Yaskawa INFORM job: DEMO_ROOF_SIDE_0625_3PAINT_3.JBI

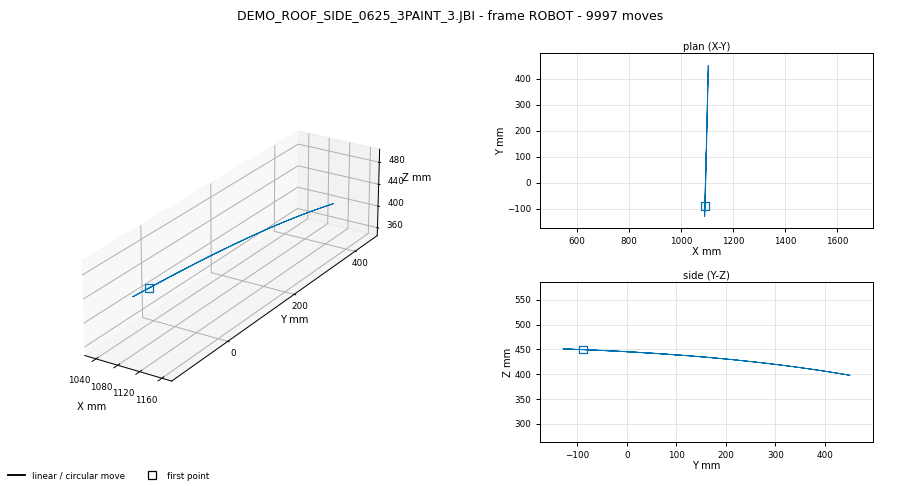
[picture p0: tool path of DEMO_ROOF_SIDE_0625_3PAINT_3.JBI in frame ROBOT, 9997 of 9997 moves have a stored position in this frame; points joined in program order, loops and branches not executed]
/JOB
//NAME DEMO_ROOF_SIDE_0625_3PAINT3
//POS
///NPOS 9997,0,0,0,0,0
///TOOL 0
///USER 0
///POSTYPE ROBOT
///RECTAN
///RCONF 1,0,0,0,0,0,0,0,0,0,0,0,0,0,0,0,0,0,0,0,0,0,0,0
C00000=1093.396,-88.065,450.012,175.022,15.482,152.318
C00001=1093.401,-87.815,450.002,175.023,15.482,152.318
C00002=1093.408,-87.566,449.991,175.025,15.483,152.317
C00003=1093.413,-87.316,449.981,175.027,15.484,152.317
C00004=1093.419,-87.066,449.970,175.029,15.485,152.317
C00005=1093.425,-86.817,449.960,175.030,15.485,152.317
C00006=1093.432,-86.567,449.949,175.032,15.486,152.317
C00007=1093.438,-86.317,449.939,175.033,15.487,152.316
C00008=1093.444,-86.068,449.928,175.035,15.487,152.316
C00009=1093.449,-85.818,449.918,175.037,15.488,152.316
C00010=1093.456,-85.568,449.908,175.038,15.488,152.316
C00011=1093.462,-85.318,449.897,175.040,15.489,152.316
C00012=1093.468,-85.069,449.886,175.042,15.490,152.315
C00013=1093.474,-84.819,449.876,175.044,15.491,152.315
C00014=1093.480,-84.569,449.865,175.045,15.491,152.315
C00015=1093.486,-84.320,449.855,175.046,15.492,152.315
C00016=1093.492,-84.070,449.844,175.048,15.493,152.315
C00017=1093.499,-83.820,449.834,175.050,15.493,152.314
C00018=1093.504,-83.571,449.823,175.052,15.494,152.314
C00019=1093.510,-83.321,449.813,175.053,15.495,152.314
C00020=1093.517,-83.071,449.803,175.055,15.495,152.314
C00021=1093.523,-82.821,449.792,175.057,15.496,152.313
C00022=1093.528,-82.572,449.781,175.059,15.497,152.313
C00023=1093.535,-82.322,449.771,175.060,15.498,152.313
C00024=1093.541,-82.072,449.759,175.061,15.498,152.313
C00025=1093.547,-81.822,449.750,175.063,15.499,152.313
C00026=1093.553,-81.573,449.739,175.065,15.499,152.312
C00027=1093.559,-81.323,449.728,175.067,15.500,152.312
C00028=1093.566,-81.050,449.716,175.069,15.501,152.312
C00029=1093.573,-80.778,449.704,175.070,15.502,152.312
C00030=1093.579,-80.506,449.693,175.072,15.502,152.311
C00031=1093.585,-80.233,449.682,175.074,15.504,152.311
C00032=1093.591,-79.984,449.671,175.075,15.504,152.311
C00033=1093.598,-79.734,449.660,175.077,15.504,152.311
C00034=1093.604,-79.484,449.650,175.079,15.505,152.311
C00035=1093.610,-79.235,449.639,175.080,15.506,152.310
C00036=1093.615,-78.985,449.628,175.082,15.507,152.310
C00037=1093.621,-78.734,449.617,175.084,15.508,152.310
C00038=1093.628,-78.485,449.607,175.085,15.508,152.310
C00039=1093.634,-78.236,449.596,175.087,15.509,152.310
C00040=1093.639,-77.986,449.585,175.088,15.510,152.309
C00041=1093.646,-77.736,449.574,175.090,15.511,152.309
C00042=1093.652,-77.487,449.563,175.092,15.511,152.309
C00043=1093.657,-77.236,449.553,175.094,15.513,152.309
C00044=1093.663,-76.987,449.543,175.095,15.513,152.309
C00045=1093.670,-76.737,449.531,175.097,15.513,152.308
C00046=1093.676,-76.488,449.521,175.098,15.515,152.308
C00047=1093.681,-76.238,449.510,175.100,15.515,152.308
C00048=1093.687,-75.989,449.499,175.102,15.516,152.308
C00049=1093.693,-75.738,449.488,175.104,15.517,152.308
C00050=1093.700,-75.489,449.477,175.105,15.517,152.307
C00051=1093.706,-75.240,449.466,175.106,15.518,152.307
C00052=1093.712,-74.990,449.455,175.108,15.519,152.307
C00053=1093.718,-74.740,449.444,175.110,15.520,152.307
C00054=1093.723,-74.491,449.433,175.112,15.521,152.307
C00055=1093.729,-74.241,449.422,175.114,15.522,152.306
C00056=1093.735,-73.991,449.411,175.116,15.522,152.306
C00057=1093.741,-73.741,449.401,175.116,15.523,152.306
C00058=1093.747,-73.491,449.390,175.118,15.523,152.306
C00059=1093.752,-73.242,449.379,175.120,15.525,152.306
C00060=1093.759,-72.992,449.368,175.122,15.525,152.305
C00061=1093.764,-72.742,449.357,175.123,15.526,152.305
C00062=1093.770,-72.493,449.346,175.125,15.527,152.305
C00063=1093.776,-72.243,449.335,175.127,15.528,152.305
C00064=1093.782,-71.993,449.324,175.128,15.528,152.305
C00065=1093.788,-71.743,449.313,175.130,15.530,152.305
C00066=1093.794,-71.494,449.302,175.132,15.530,152.304
C00067=1093.799,-71.245,449.292,175.133,15.531,152.304
C00068=1093.806,-70.994,449.280,175.135,15.532,152.304
C00069=1093.812,-70.745,449.269,175.137,15.533,152.304
C00070=1093.818,-70.496,449.258,175.138,15.534,152.304
C00071=1093.824,-70.246,449.247,175.140,15.535,152.303
C00072=1093.830,-69.996,449.236,175.141,15.535,152.303
C00073=1093.835,-69.746,449.224,175.143,15.536,152.303
C00074=1093.840,-69.497,449.213,175.145,15.537,152.303
C00075=1093.847,-69.247,449.202,175.147,15.538,152.303
C00076=1093.853,-68.997,449.191,175.148,15.539,152.303
C00077=1093.858,-68.748,449.180,175.150,15.540,152.302
C00078=1093.865,-68.498,449.169,175.152,15.541,152.302
C00079=1093.870,-68.248,449.158,175.154,15.541,152.302
C00080=1093.876,-67.999,449.147,175.155,15.543,152.302
C00081=1093.882,-67.748,449.136,175.156,15.543,152.302
C00082=1093.888,-67.500,449.125,175.158,15.543,152.301
C00083=1093.894,-67.250,449.114,175.160,15.545,152.301
C00084=1093.900,-67.000,449.102,175.162,15.545,152.301
C00085=1093.906,-66.750,449.091,175.163,15.546,152.301
C00086=1093.911,-66.501,449.080,175.165,15.547,152.301
C00087=1093.918,-66.250,449.069,175.167,15.548,152.300
C00088=1093.923,-66.001,449.058,175.169,15.549,152.300
C00089=1093.929,-65.752,449.046,175.170,15.550,152.300
C00090=1093.936,-65.502,449.035,175.171,15.550,152.300
C00091=1093.941,-65.252,449.024,175.173,15.551,152.300
C00092=1093.948,-64.982,449.012,175.175,15.552,152.300
C00093=1093.954,-64.711,449.000,175.177,15.554,152.299
C00094=1093.960,-64.441,448.988,175.179,15.555,152.299
C00095=1093.967,-64.171,448.975,175.181,15.555,152.299
C00096=1093.972,-63.921,448.964,175.182,15.556,152.299
C00097=1093.979,-63.672,448.952,175.184,15.556,152.299
C00098=1093.985,-63.422,448.942,175.185,15.558,152.298
C00099=1093.991,-63.172,448.930,175.187,15.558,152.298
C00100=1093.997,-62.922,448.919,175.189,15.559,152.298
C00101=1094.002,-62.673,448.907,175.191,15.560,152.298
C00102=1094.009,-62.423,448.896,175.192,15.561,152.298
C00103=1094.014,-62.174,448.885,175.194,15.562,152.297
C00104=1094.021,-61.923,448.874,175.196,15.563,152.297
C00105=1094.027,-61.674,448.862,175.198,15.564,152.297
C00106=1094.033,-61.424,448.851,175.199,15.565,152.297
C00107=1094.038,-61.174,448.840,175.201,15.566,152.297
C00108=1094.044,-60.926,448.828,175.203,15.567,152.297
C00109=1094.050,-60.675,448.817,175.204,15.567,152.296
C00110=1094.056,-60.426,448.806,175.205,15.568,152.296
C00111=1094.063,-60.176,448.795,175.207,15.569,152.296
C00112=1094.068,-59.927,448.782,175.209,15.570,152.296
C00113=1094.074,-59.676,448.771,175.211,15.571,152.296
C00114=1094.080,-59.427,448.760,175.213,15.571,152.295
C00115=1094.087,-59.177,448.748,175.214,15.573,152.295
C00116=1094.092,-58.928,448.738,175.216,15.573,152.295
C00117=1094.098,-58.677,448.726,175.218,15.574,152.295
C00118=1094.104,-58.428,448.714,175.220,15.575,152.295
C00119=1094.110,-58.178,448.703,175.221,15.576,152.295
C00120=1094.116,-57.929,448.691,175.223,15.577,152.294
C00121=1094.123,-57.679,448.680,175.225,15.578,152.294
C00122=1094.128,-57.429,448.669,175.226,15.579,152.294
C00123=1094.134,-57.181,448.657,175.228,15.580,152.294
C00124=1094.140,-56.930,448.646,175.230,15.581,152.294
C00125=1094.147,-56.681,448.634,175.231,15.581,152.294
C00126=1094.152,-56.431,448.622,175.233,15.582,152.293
C00127=1094.158,-56.181,448.611,175.234,15.583,152.293
C00128=1094.164,-55.932,448.599,175.236,15.584,152.293
C00129=1094.170,-55.682,448.588,175.238,15.585,152.293
C00130=1094.176,-55.433,448.576,175.240,15.586,152.293
C00131=1094.182,-55.182,448.565,175.241,15.587,152.292
C00132=1094.188,-54.933,448.553,175.243,15.588,152.292
C00133=1094.194,-54.683,448.542,175.245,15.589,152.292
C00134=1094.200,-54.434,448.530,175.247,15.589,152.292
C00135=1094.206,-54.184,448.519,175.248,15.590,152.292
C00136=1094.212,-53.935,448.507,175.250,15.591,152.291
C00137=1094.218,-53.685,448.496,175.252,15.592,152.291
C00138=1094.224,-53.436,448.483,175.254,15.593,152.291
C00139=1094.230,-53.185,448.472,175.255,15.594,152.291
C00140=1094.237,-52.936,448.460,175.257,15.595,152.291
C00141=1094.243,-52.686,448.449,175.259,15.596,152.290
C00142=1094.248,-52.437,448.437,175.261,15.597,152.290
C00143=1094.254,-52.187,448.426,175.262,15.597,152.290
C00144=1094.261,-51.937,448.414,175.264,15.599,152.290
C00145=1094.266,-51.687,448.402,175.266,15.599,152.290
C00146=1094.272,-51.438,448.391,175.267,15.600,152.290
C00147=1094.279,-51.188,448.379,175.269,15.601,152.289
C00148=1094.284,-50.939,448.367,175.270,15.602,152.289
C00149=1094.291,-50.689,448.355,175.272,15.602,152.289
C00150=1094.297,-50.439,448.344,175.274,15.604,152.289
C00151=1094.302,-50.190,448.332,175.276,15.604,152.289
C00152=1094.309,-49.940,448.321,175.277,15.605,152.289
C00153=1094.314,-49.690,448.308,175.279,15.606,152.288
C00154=1094.321,-49.441,448.296,175.281,15.607,152.288
C00155=1094.326,-49.191,448.285,175.282,15.609,152.288
C00156=1094.332,-48.922,448.272,175.285,15.610,152.288
C00157=1094.338,-48.653,448.259,175.286,15.611,152.288
C00158=1094.345,-48.384,448.247,175.288,15.612,152.287
C00159=1094.351,-48.115,448.234,175.290,15.613,152.287
C00160=1094.357,-47.866,448.222,175.292,15.613,152.287
C00161=1094.363,-47.615,448.211,175.293,15.615,152.287
C00162=1094.368,-47.366,448.198,175.295,15.615,152.287
C00163=1094.375,-47.117,448.187,175.297,15.617,152.287
C00164=1094.381,-46.866,448.175,175.299,15.618,152.286
C00165=1094.386,-46.617,448.162,175.300,15.618,152.286
C00166=1094.393,-46.367,448.151,175.302,15.620,152.286
C00167=1094.398,-46.118,448.138,175.304,15.620,152.286
C00168=1094.404,-45.868,448.127,175.305,15.621,152.286
C00169=1094.410,-45.618,448.115,175.307,15.622,152.286
C00170=1094.416,-45.369,448.103,175.309,15.623,152.285
C00171=1094.422,-45.119,448.091,175.311,15.624,152.285
C00172=1094.427,-44.870,448.079,175.312,15.625,152.285
C00173=1094.434,-44.620,448.067,175.314,15.626,152.285
C00174=1094.440,-44.370,448.054,175.316,15.627,152.285
C00175=1094.445,-44.121,448.044,175.318,15.628,152.285
C00176=1094.451,-43.871,448.031,175.319,15.629,152.284
C00177=1094.457,-43.622,448.019,175.321,15.630,152.284
C00178=1094.463,-43.372,448.007,175.323,15.631,152.284
C00179=1094.469,-43.122,447.995,175.324,15.632,152.284
C00180=1094.475,-42.873,447.983,175.326,15.633,152.284
C00181=1094.481,-42.623,447.971,175.328,15.634,152.284
C00182=1094.487,-42.373,447.959,175.330,15.635,152.283
C00183=1094.492,-42.123,447.947,175.331,15.636,152.283
C00184=1094.498,-41.874,447.935,175.333,15.637,152.283
C00185=1094.504,-41.625,447.923,175.335,15.638,152.283
C00186=1094.510,-41.375,447.911,175.337,15.639,152.283
C00187=1094.516,-41.125,447.898,175.338,15.640,152.283
C00188=1094.522,-40.876,447.887,175.340,15.641,152.282
C00189=1094.528,-40.626,447.875,175.342,15.642,152.282
C00190=1094.535,-40.376,447.863,175.343,15.642,152.282
C00191=1094.540,-40.126,447.850,175.345,15.644,152.282
C00192=1094.546,-39.877,447.838,175.347,15.644,152.282
C00193=1094.552,-39.627,447.826,175.349,15.645,152.281
C00194=1094.558,-39.377,447.814,175.351,15.647,152.281
C00195=1094.564,-39.128,447.801,175.353,15.648,152.281
C00196=1094.570,-38.878,447.790,175.354,15.649,152.281
C00197=1094.576,-38.628,447.778,175.356,15.650,152.281
C00198=1094.581,-38.379,447.765,175.358,15.651,152.281
C00199=1094.587,-38.129,447.753,175.360,15.652,152.280
C00200=1094.594,-37.880,447.741,175.361,15.653,152.280
C00201=1094.599,-37.630,447.729,175.363,15.654,152.280
C00202=1094.605,-37.381,447.716,175.365,15.655,152.280
C00203=1094.611,-37.131,447.704,175.366,15.656,152.280
C00204=1094.616,-36.881,447.691,175.368,15.657,152.280
C00205=1094.622,-36.632,447.679,175.370,15.658,152.279
C00206=1094.629,-36.382,447.667,175.372,15.659,152.279
C00207=1094.634,-36.133,447.655,175.373,15.659,152.279
C00208=1094.640,-35.883,447.642,175.375,15.661,152.279
C00209=1094.646,-35.633,447.630,175.377,15.662,152.279
C00210=1094.651,-35.384,447.617,175.378,15.663,152.279
C00211=1094.658,-35.134,447.605,175.380,15.664,152.279
C00212=1094.664,-34.884,447.593,175.382,15.664,152.278
C00213=1094.669,-34.635,447.581,175.384,15.666,152.278
C00214=1094.675,-34.385,447.568,175.386,15.667,152.278
C00215=1094.681,-34.135,447.556,175.388,15.668,152.278
C00216=1094.687,-33.886,447.543,175.389,15.669,152.278
C00217=1094.692,-33.636,447.531,175.391,15.670,152.277
C00218=1094.699,-33.387,447.519,175.393,15.671,152.277
C00219=1094.705,-33.137,447.506,175.394,15.672,152.277
C00220=1094.711,-32.868,447.493,175.396,15.673,152.277
C00221=1094.718,-32.600,447.479,175.398,15.674,152.277
C00222=1094.722,-32.331,447.467,175.401,15.675,152.277
C00223=1094.729,-32.062,447.453,175.402,15.677,152.276
C00224=1094.735,-31.812,447.441,175.404,15.677,152.276
C00225=1094.742,-31.563,447.428,175.406,15.678,152.276
C00226=1094.748,-31.313,447.415,175.407,15.680,152.276
C00227=1094.753,-31.064,447.403,175.409,15.680,152.276
C00228=1094.759,-30.814,447.391,175.411,15.681,152.276
C00229=1094.765,-30.564,447.378,175.413,15.682,152.275
C00230=1094.771,-30.315,447.366,175.414,15.683,152.275
C00231=1094.777,-30.065,447.353,175.416,15.684,152.275
C00232=1094.782,-29.816,447.341,175.419,15.686,152.275
C00233=1094.788,-29.566,447.328,175.420,15.687,152.275
C00234=1094.794,-29.316,447.315,175.422,15.688,152.275
C00235=1094.801,-29.067,447.303,175.424,15.689,152.274
C00236=1094.807,-28.817,447.290,175.426,15.689,152.274
C00237=1094.812,-28.568,447.278,175.427,15.691,152.274
C00238=1094.818,-28.318,447.266,175.429,15.692,152.274
C00239=1094.824,-28.069,447.252,175.431,15.693,152.274
C00240=1094.830,-27.819,447.240,175.432,15.694,152.274
C00241=1094.836,-27.569,447.227,175.434,15.694,152.273
C00242=1094.841,-27.320,447.215,175.436,15.696,152.273
C00243=1094.847,-27.070,447.203,175.438,15.696,152.273
C00244=1094.853,-26.820,447.189,175.440,15.698,152.273
C00245=1094.859,-26.571,447.177,175.442,15.699,152.273
C00246=1094.865,-26.321,447.164,175.443,15.700,152.272
C00247=1094.870,-26.072,447.152,175.445,15.701,152.272
C00248=1094.877,-25.822,447.139,175.447,15.702,152.272
C00249=1094.882,-25.572,447.126,175.448,15.703,152.272
C00250=1094.888,-25.323,447.114,175.450,15.704,152.272
C00251=1094.894,-25.072,447.101,175.452,15.705,152.272
C00252=1094.899,-24.824,447.088,175.454,15.706,152.272
C00253=1094.905,-24.574,447.075,175.456,15.708,152.271
C00254=1094.911,-24.324,447.063,175.458,15.708,152.271
C00255=1094.917,-24.074,447.050,175.459,15.710,152.271
C00256=1094.923,-23.825,447.037,175.461,15.710,152.271
C00257=1094.929,-23.575,447.024,175.463,15.711,152.271
C00258=1094.934,-23.326,447.012,175.464,15.713,152.271
C00259=1094.940,-23.077,446.999,175.466,15.713,152.270
C00260=1094.946,-22.826,446.986,175.468,15.714,152.270
C00261=1094.952,-22.576,446.973,175.470,15.715,152.270
C00262=1094.958,-22.327,446.960,175.472,15.717,152.270
C00263=1094.964,-22.077,446.947,175.474,15.718,152.270
C00264=1094.969,-21.828,446.935,175.476,15.719,152.270
C00265=1094.975,-21.579,446.922,175.477,15.720,152.269
C00266=1094.981,-21.329,446.909,175.479,15.721,152.269
C00267=1094.987,-21.079,446.895,175.481,15.722,152.269
C00268=1094.993,-20.829,446.883,175.482,15.723,152.269
C00269=1094.998,-20.580,446.870,175.484,15.724,152.269
C00270=1095.005,-20.330,446.857,175.487,15.725,152.269
C00271=1095.011,-20.080,446.844,175.489,15.726,152.268
C00272=1095.016,-19.832,446.831,175.490,15.727,152.268
C00273=1095.021,-19.582,446.818,175.492,15.729,152.268
C00274=1095.027,-19.332,446.806,175.494,15.729,152.268
C00275=1095.033,-19.083,446.792,175.495,15.730,152.268
C00276=1095.039,-18.833,446.780,175.497,15.731,152.267
C00277=1095.046,-18.583,446.767,175.499,15.732,152.267
C00278=1095.051,-18.334,446.754,175.501,15.734,152.267
C00279=1095.057,-18.084,446.740,175.503,15.735,152.267
C00280=1095.063,-17.834,446.728,175.505,15.736,152.267
C00281=1095.069,-17.585,446.714,175.506,15.737,152.267
C00282=1095.075,-17.335,446.702,175.508,15.738,152.267
C00283=1095.081,-17.086,446.689,175.510,15.738,152.266
C00284=1095.087,-16.817,446.675,175.512,15.740,152.266
C00285=1095.093,-16.547,446.660,175.514,15.741,152.266
C00286=1095.100,-16.277,446.646,175.516,15.742,152.266
C00287=1095.106,-16.007,446.632,175.518,15.743,152.266
C00288=1095.112,-15.758,446.619,175.520,15.745,152.265
C00289=1095.118,-15.509,446.606,175.522,15.745,152.265
C00290=1095.124,-15.259,446.593,175.524,15.746,152.265
C00291=1095.129,-15.010,446.580,175.525,15.747,152.265
C00292=1095.135,-14.760,446.567,175.527,15.748,152.265
C00293=1095.141,-14.511,446.554,175.529,15.749,152.265
C00294=1095.146,-14.260,446.541,175.531,15.751,152.264
C00295=1095.152,-14.011,446.527,175.533,15.752,152.264
C00296=1095.159,-13.762,446.514,175.535,15.753,152.264
C00297=1095.164,-13.512,446.501,175.536,15.754,152.264
C00298=1095.170,-13.262,446.488,175.538,15.755,152.264
C00299=1095.175,-13.012,446.475,175.540,15.756,152.263
C00300=1095.181,-12.763,446.461,175.541,15.757,152.263
C00301=1095.188,-12.514,446.448,175.544,15.758,152.263
C00302=1095.193,-12.264,446.435,175.546,15.759,152.263
C00303=1095.199,-12.014,446.422,175.547,15.760,152.263
C00304=1095.204,-11.765,446.408,175.549,15.761,152.263
C00305=1095.210,-11.515,446.395,175.551,15.762,152.263
C00306=1095.217,-11.266,446.382,175.553,15.763,152.262
C00307=1095.222,-11.016,446.368,175.555,15.765,152.262
C00308=1095.228,-10.766,446.356,175.557,15.765,152.262
C00309=1095.233,-10.516,446.342,175.559,15.767,152.262
C00310=1095.240,-10.267,446.328,175.560,15.768,152.262
C00311=1095.245,-10.017,446.315,175.562,15.768,152.261
C00312=1095.251,-9.768,446.302,175.564,15.770,152.261
C00313=1095.257,-9.519,446.289,175.566,15.771,152.261
C00314=1095.262,-9.268,446.276,175.568,15.772,152.261
C00315=1095.269,-9.019,446.262,175.570,15.773,152.261
C00316=1095.274,-8.769,446.248,175.571,15.774,152.261
C00317=1095.280,-8.520,446.235,175.573,15.775,152.260
C00318=1095.285,-8.270,446.222,175.576,15.776,152.260
C00319=1095.292,-8.021,446.209,175.577,15.778,152.260
C00320=1095.297,-7.771,446.195,175.579,15.778,152.260
C00321=1095.303,-7.522,446.182,175.581,15.779,152.260
C00322=1095.309,-7.272,446.168,175.583,15.780,152.259
C00323=1095.315,-7.022,446.155,175.584,15.781,152.259
C00324=1095.321,-6.773,446.142,175.587,15.783,152.259
C00325=1095.326,-6.524,446.128,175.588,15.784,152.259
C00326=1095.333,-6.274,446.115,175.590,15.785,152.259
C00327=1095.338,-6.025,446.101,175.592,15.786,152.259
C00328=1095.344,-5.775,446.088,175.594,15.786,152.258
C00329=1095.350,-5.525,446.075,175.595,15.788,152.258
C00330=1095.356,-5.276,446.061,175.598,15.789,152.258
C00331=1095.362,-5.026,446.047,175.600,15.790,152.258
C00332=1095.368,-4.777,446.034,175.602,15.791,152.258
C00333=1095.373,-4.527,446.020,175.603,15.792,152.258
C00334=1095.380,-4.278,446.007,175.605,15.793,152.257
C00335=1095.385,-4.028,445.993,175.607,15.794,152.257
C00336=1095.391,-3.778,445.980,175.609,15.795,152.257
C00337=1095.397,-3.529,445.966,175.611,15.796,152.257
C00338=1095.402,-3.279,445.952,175.613,15.797,152.257
C00339=1095.408,-3.030,445.939,175.614,15.798,152.256
C00340=1095.414,-2.780,445.925,175.617,15.799,152.256
C00341=1095.419,-2.531,445.911,175.619,15.801,152.256
C00342=1095.425,-2.281,445.898,175.620,15.802,152.256
C00343=1095.431,-2.031,445.884,175.622,15.802,152.256
C00344=1095.437,-1.782,445.870,175.624,15.804,152.256
C00345=1095.442,-1.532,445.856,175.626,15.805,152.255
C00346=1095.449,-1.283,445.843,175.628,15.806,152.255
C00347=1095.454,-1.033,445.829,175.630,15.807,152.255
C00348=1095.460,-0.762,445.815,175.631,15.808,152.255
C00349=1095.466,-0.491,445.799,175.634,15.809,152.255
C00350=1095.472,-0.220,445.785,175.636,15.810,152.254
C00351=1095.478,0.052,445.770,175.638,15.812,152.254
C00352=1095.485,0.302,445.756,175.640,15.813,152.254
C00353=1095.490,0.551,445.743,175.642,15.814,152.254
C00354=1095.496,0.801,445.729,175.644,15.815,152.254
C00355=1095.502,1.050,445.714,175.646,15.816,152.254
C00356=1095.508,1.299,445.701,175.648,15.817,152.253
C00357=1095.513,1.548,445.687,175.649,15.818,152.253
C00358=1095.519,1.798,445.673,175.651,15.819,152.253
C00359=1095.524,2.048,445.659,175.653,15.820,152.253
C00360=1095.530,2.297,445.646,175.656,15.821,152.253
C00361=1095.536,2.547,445.632,175.657,15.823,152.252
C00362=1095.542,2.797,445.618,175.659,15.823,152.252
C00363=1095.547,3.046,445.604,175.661,15.825,152.252
C00364=1095.553,3.296,445.590,175.663,15.826,152.252
C00365=1095.559,3.545,445.577,175.665,15.827,152.252
C00366=1095.565,3.795,445.563,175.667,15.828,152.252
C00367=1095.571,4.045,445.549,175.668,15.829,152.251
C00368=1095.576,4.294,445.534,175.670,15.830,152.251
C00369=1095.582,4.544,445.520,175.673,15.831,152.251
C00370=1095.588,4.793,445.507,175.675,15.832,152.251
C00371=1095.594,5.042,445.493,175.676,15.833,152.251
C00372=1095.599,5.292,445.479,175.678,15.834,152.250
C00373=1095.605,5.542,445.465,175.681,15.835,152.250
C00374=1095.611,5.791,445.450,175.682,15.836,152.250
C00375=1095.617,6.040,445.437,175.684,15.837,152.250
C00376=1095.623,6.290,445.423,175.686,15.838,152.250
C00377=1095.628,6.540,445.409,175.688,15.840,152.249
C00378=1095.634,6.790,445.395,175.690,15.841,152.249
C00379=1095.640,7.039,445.381,175.692,15.841,152.249
C00380=1095.645,7.288,445.367,175.694,15.843,152.249
C00381=1095.652,7.538,445.354,175.695,15.843,152.249
C00382=1095.658,7.788,445.339,175.698,15.845,152.248
C00383=1095.664,8.037,445.325,175.700,15.846,152.248
C00384=1095.669,8.286,445.311,175.702,15.846,152.248
C00385=1095.674,8.536,445.297,175.703,15.848,152.248
C00386=1095.680,8.786,445.283,175.706,15.849,152.248
C00387=1095.686,9.035,445.268,175.707,15.850,152.248
C00388=1095.692,9.285,445.254,175.709,15.851,152.247
C00389=1095.698,9.534,445.241,175.711,15.851,152.247
C00390=1095.704,9.784,445.227,175.714,15.853,152.247
C00391=1095.710,10.033,445.212,175.715,15.854,152.247
C00392=1095.715,10.283,445.198,175.717,15.855,152.246
C00393=1095.721,10.532,445.185,175.719,15.856,152.246
C00394=1095.727,10.782,445.170,175.722,15.857,152.246
C00395=1095.733,11.032,445.156,175.723,15.858,152.246
C00396=1095.738,11.281,445.142,175.725,15.859,152.246
C00397=1095.745,11.531,445.127,175.727,15.860,152.245
C00398=1095.751,11.780,445.114,175.729,15.861,152.245
C00399=1095.757,12.029,445.099,175.731,15.862,152.245
C00400=1095.762,12.279,445.085,175.733,15.863,152.245
C00401=1095.768,12.529,445.071,175.735,15.864,152.245
C00402=1095.774,12.778,445.056,175.737,15.865,152.244
C00403=1095.779,13.028,445.043,175.739,15.866,152.244
C00404=1095.786,13.277,445.028,175.741,15.867,152.244
C00405=1095.791,13.527,445.014,175.743,15.868,152.244
C00406=1095.797,13.776,445.000,175.745,15.870,152.244
C00407=1095.803,14.026,444.985,175.747,15.870,152.243
C00408=1095.809,14.276,444.971,175.749,15.871,152.243
C00409=1095.814,14.525,444.956,175.751,15.872,152.243
C00410=1095.820,14.775,444.942,175.753,15.873,152.243
C00411=1095.826,15.024,444.928,175.755,15.874,152.243
C00412=1095.833,15.297,444.912,175.757,15.875,152.242
C00413=1095.839,15.571,444.897,175.759,15.877,152.242
C00414=1095.845,15.844,444.881,175.761,15.877,152.242
C00415=1095.851,16.117,444.865,175.764,15.879,152.242
C00416=1095.857,16.366,444.850,175.766,15.880,152.241
C00417=1095.863,16.615,444.836,175.767,15.880,152.241
C00418=1095.869,16.865,444.821,175.770,15.882,152.241
C00419=1095.874,17.114,444.807,175.772,15.883,152.241
C00420=1095.880,17.363,444.793,175.774,15.884,152.241
C00421=1095.886,17.614,444.779,175.776,15.885,152.240
C00422=1095.891,17.863,444.763,175.778,15.886,152.240
C00423=1095.897,18.113,444.750,175.780,15.887,152.240
C00424=1095.903,18.362,444.735,175.781,15.888,152.240
C00425=1095.909,18.612,444.721,175.784,15.889,152.240
C00426=1095.915,18.861,444.706,175.786,15.890,152.239
C00427=1095.921,19.110,444.691,175.788,15.891,152.239
C00428=1095.926,19.360,444.677,175.789,15.892,152.239
C00429=1095.932,19.610,444.662,175.792,15.893,152.239
C00430=1095.937,19.859,444.648,175.794,15.894,152.239
C00431=1095.943,20.108,444.633,175.796,15.895,152.238
C00432=1095.950,20.358,444.618,175.798,15.896,152.238
C00433=1095.955,20.608,444.605,175.800,15.897,152.238
C00434=1095.961,20.858,444.589,175.802,15.898,152.238
C00435=1095.966,21.107,444.574,175.804,15.899,152.237
C00436=1095.972,21.356,444.561,175.806,15.901,152.237
C00437=1095.978,21.606,444.546,175.808,15.901,152.237
C00438=1095.983,21.855,444.530,175.810,15.902,152.237
C00439=1095.989,22.105,444.517,175.812,15.904,152.237
C00440=1095.995,22.354,444.502,175.814,15.904,152.236
C00441=1096.001,22.603,444.487,175.816,15.905,152.236
C00442=1096.006,22.854,444.472,175.819,15.906,152.236
C00443=1096.012,23.103,444.458,175.820,15.908,152.236
C00444=1096.019,23.352,444.443,175.822,15.908,152.236
C00445=1096.024,23.601,444.428,175.824,15.909,152.235
C00446=1096.029,23.851,444.414,175.826,15.911,152.235
C00447=1096.035,24.101,444.399,175.828,15.911,152.235
C00448=1096.041,24.350,444.384,175.830,15.912,152.235
C00449=1096.047,24.600,444.369,175.833,15.913,152.234
C00450=1096.052,24.849,444.355,175.834,15.915,152.234
C00451=1096.059,25.099,444.340,175.836,15.915,152.234
C00452=1096.064,25.348,444.325,175.839,15.917,152.234
C00453=1096.070,25.597,444.310,175.841,15.917,152.233
C00454=1096.076,25.847,444.295,175.842,15.918,152.233
C00455=1096.081,26.097,444.281,175.844,15.919,152.233
C00456=1096.087,26.347,444.266,175.847,15.920,152.233
C00457=1096.093,26.596,444.251,175.849,15.921,152.233
C00458=1096.099,26.845,444.236,175.851,15.922,152.232
C00459=1096.104,27.094,444.221,175.853,15.924,152.232
C00460=1096.111,27.344,444.206,175.855,15.924,152.232
C00461=1096.115,27.594,444.192,175.857,15.925,152.232
C00462=1096.122,27.844,444.177,175.860,15.926,152.231
C00463=1096.128,28.093,444.162,175.861,15.927,152.231
C00464=1096.133,28.343,444.147,175.863,15.928,152.231
C00465=1096.139,28.592,444.132,175.866,15.929,152.231
C00466=1096.145,28.841,444.117,175.868,15.930,152.231
C00467=1096.150,29.090,444.102,175.870,15.931,152.230
C00468=1096.157,29.340,444.087,175.872,15.933,152.230
C00469=1096.162,29.589,444.072,175.874,15.933,152.230
C00470=1096.168,29.839,444.057,175.876,15.934,152.230
C00471=1096.173,30.088,444.042,175.878,15.935,152.229
C00472=1096.179,30.339,444.027,175.880,15.936,152.229
C00473=1096.184,30.588,444.012,175.882,15.937,152.229
C00474=1096.191,30.837,443.997,175.885,15.939,152.229
C00475=1096.196,31.087,443.982,175.887,15.939,152.228
C00476=1096.202,31.361,443.965,175.888,15.940,152.228
C00477=1096.209,31.636,443.949,175.891,15.941,152.228
C00478=1096.215,31.910,443.932,175.894,15.942,152.228
C00479=1096.222,32.184,443.915,175.896,15.943,152.227
C00480=1096.227,32.434,443.900,175.897,15.944,152.227
C00481=1096.233,32.683,443.885,175.900,15.946,152.227
C00482=1096.239,32.933,443.870,175.902,15.946,152.227
C00483=1096.244,33.182,443.855,175.904,15.947,152.227
C00484=1096.250,33.432,443.840,175.906,15.948,152.226
C00485=1096.255,33.681,443.824,175.908,15.949,152.226
C00486=1096.262,33.931,443.810,175.910,15.950,152.226
C00487=1096.267,34.180,443.794,175.913,15.951,152.226
C00488=1096.273,34.430,443.779,175.914,15.952,152.225
C00489=1096.279,34.680,443.764,175.916,15.953,152.225
C00490=1096.284,34.929,443.749,175.919,15.954,152.225
C00491=1096.290,35.179,443.734,175.921,15.955,152.225
C00492=1096.296,35.428,443.719,175.923,15.956,152.224
C00493=1096.302,35.677,443.703,175.925,15.957,152.224
C00494=1096.307,35.927,443.687,175.927,15.958,152.224
C00495=1096.313,36.176,443.673,175.929,15.959,152.224
C00496=1096.319,36.426,443.657,175.932,15.960,152.223
C00497=1096.325,36.675,443.643,175.934,15.961,152.223
C00498=1096.330,36.925,443.627,175.936,15.962,152.223
C00499=1096.336,37.175,443.612,175.938,15.963,152.223
C00500=1096.342,37.423,443.596,175.940,15.963,152.222
C00501=1096.348,37.673,443.581,175.943,15.965,152.222
C00502=1096.353,37.922,443.566,175.945,15.965,152.222
C00503=1096.359,38.172,443.551,175.946,15.966,152.222
C00504=1096.365,38.422,443.535,175.949,15.967,152.221
C00505=1096.371,38.670,443.520,175.951,15.968,152.221
C00506=1096.376,38.920,443.504,175.953,15.969,152.221
C00507=1096.382,39.170,443.489,175.956,15.970,152.220
C00508=1096.387,39.420,443.474,175.957,15.971,152.220
C00509=1096.394,39.669,443.458,175.959,15.972,152.220
C00510=1096.399,39.918,443.443,175.962,15.973,152.220
C00511=1096.405,40.168,443.427,175.964,15.974,152.220
C00512=1096.410,40.417,443.412,175.966,15.975,152.219
C00513=1096.416,40.666,443.396,175.968,15.976,152.219
C00514=1096.422,40.916,443.381,175.970,15.977,152.219
C00515=1096.427,41.165,443.366,175.973,15.978,152.219
C00516=1096.433,41.415,443.349,175.975,15.979,152.218
C00517=1096.439,41.664,443.334,175.977,15.979,152.218
C00518=1096.444,41.914,443.319,175.979,15.981,152.218
C00519=1096.450,42.163,443.303,175.981,15.981,152.217
C00520=1096.456,42.413,443.287,175.983,15.982,152.217
C00521=1096.461,42.662,443.272,175.986,15.983,152.217
C00522=1096.468,42.911,443.257,175.988,15.984,152.217
C00523=1096.473,43.161,443.241,175.990,15.985,152.216
C00524=1096.478,43.410,443.226,175.992,15.986,152.216
C00525=1096.484,43.660,443.210,175.994,15.987,152.216
C00526=1096.490,43.910,443.194,175.997,15.988,152.216
C00527=1096.495,44.158,443.178,175.999,15.989,152.215
C00528=1096.502,44.408,443.163,176.000,15.989,152.215
C00529=1096.507,44.658,443.148,176.003,15.991,152.215
C00530=1096.513,44.907,443.132,176.005,15.991,152.215
C00531=1096.518,45.157,443.116,176.008,15.993,152.214
C00532=1096.524,45.406,443.100,176.010,15.993,152.214
C00533=1096.529,45.655,443.085,176.012,15.994,152.214
C00534=1096.535,45.905,443.069,176.014,15.995,152.214
C00535=1096.541,46.155,443.053,176.016,15.996,152.213
C00536=1096.546,46.403,443.037,176.018,15.997,152.213
C00537=1096.552,46.653,443.022,176.021,15.998,152.213
C00538=1096.558,46.903,443.006,176.023,15.999,152.213
C00539=1096.563,47.152,442.990,176.025,16.000,152.212
C00540=1096.569,47.427,442.972,176.027,16.001,152.212
C00541=1096.575,47.701,442.955,176.030,16.002,152.212
C00542=1096.582,47.976,442.938,176.032,16.003,152.211
C00543=1096.587,48.250,442.921,176.034,16.004,152.211
C00544=1096.593,48.500,442.904,176.037,16.005,152.211
C00545=1096.599,48.750,442.889,176.039,16.006,152.211
C00546=1096.605,48.999,442.873,176.041,16.006,152.210
C00547=1096.610,49.248,442.858,176.044,16.008,152.210
C00548=1096.616,49.498,442.841,176.046,16.008,152.210
C00549=1096.622,49.747,442.825,176.048,16.010,152.209
C00550=1096.627,49.996,442.810,176.050,16.010,152.209
C00551=1096.633,50.246,442.794,176.052,16.011,152.209
C00552=1096.639,50.496,442.778,176.055,16.012,152.209
C00553=1096.645,50.745,442.762,176.057,16.013,152.208
C00554=1096.651,50.994,442.746,176.059,16.014,152.208
C00555=1096.656,51.243,442.730,176.061,16.015,152.208
C00556=1096.662,51.493,442.714,176.063,16.015,152.207
C00557=1096.667,51.742,442.698,176.066,16.017,152.207
C00558=1096.673,51.992,442.682,176.068,16.017,152.207
C00559=1096.678,52.241,442.666,176.071,16.019,152.207
C00560=1096.684,52.490,442.650,176.073,16.019,152.206
C00561=1096.689,52.740,442.634,176.075,16.020,152.206
C00562=1096.695,52.990,442.618,176.077,16.021,152.206
C00563=1096.701,53.239,442.601,176.079,16.021,152.205
C00564=1096.706,53.488,442.586,176.082,16.023,152.205
C00565=1096.712,53.738,442.570,176.084,16.023,152.205
C00566=1096.718,53.987,442.554,176.086,16.024,152.205
C00567=1096.724,54.236,442.538,176.089,16.025,152.204
C00568=1096.730,54.486,442.522,176.091,16.026,152.204
C00569=1096.736,54.736,442.506,176.093,16.027,152.204
C00570=1096.741,54.984,442.490,176.095,16.028,152.203
C00571=1096.747,55.234,442.474,176.097,16.028,152.203
C00572=1096.752,55.484,442.457,176.100,16.030,152.203
C00573=1096.758,55.733,442.441,176.102,16.030,152.202
C00574=1096.764,55.983,442.425,176.105,16.031,152.202
C00575=1096.770,56.232,442.409,176.107,16.032,152.202
C00576=1096.776,56.481,442.392,176.108,16.033,152.202
C00577=1096.782,56.731,442.376,176.111,16.033,152.201
C00578=1096.787,56.980,442.361,176.113,16.034,152.201
C00579=1096.793,57.229,442.345,176.116,16.035,152.201
C00580=1096.798,57.479,442.328,176.118,16.036,152.200
C00581=1096.804,57.728,442.312,176.121,16.037,152.200
C00582=1096.810,57.978,442.295,176.123,16.038,152.200
C00583=1096.816,58.227,442.279,176.125,16.038,152.199
C00584=1096.822,58.476,442.263,176.128,16.039,152.199
C00585=1096.828,58.726,442.247,176.130,16.040,152.199
C00586=1096.833,58.976,442.230,176.132,16.041,152.199
C00587=1096.838,59.225,442.214,176.134,16.041,152.198
C00588=1096.844,59.475,442.198,176.136,16.042,152.198
C00589=1096.850,59.723,442.182,176.139,16.043,152.197
C00590=1096.856,59.973,442.166,176.141,16.044,152.197
C00591=1096.862,60.222,442.150,176.144,16.045,152.197
C00592=1096.867,60.472,442.133,176.146,16.045,152.197
C00593=1096.873,60.721,442.116,176.149,16.047,152.196
C00594=1096.879,60.970,442.100,176.151,16.047,152.196
C00595=1096.885,61.220,442.084,176.153,16.047,152.196
C00596=1096.891,61.469,442.068,176.155,16.049,152.195
C00597=1096.896,61.719,442.051,176.158,16.049,152.195
C00598=1096.902,61.968,442.035,176.160,16.050,152.195
C00599=1096.908,62.218,442.018,176.162,16.051,152.194
C00600=1096.914,62.467,442.002,176.165,16.052,152.194
C00601=1096.919,62.717,441.985,176.167,16.053,152.194
C00602=1096.925,62.966,441.969,176.169,16.053,152.193
C00603=1096.931,63.215,441.953,176.172,16.054,152.193
C00604=1096.937,63.490,441.934,176.174,16.054,152.193
C00605=1096.944,63.764,441.916,176.177,16.056,152.192
C00606=1096.950,64.038,441.898,176.180,16.056,152.192
C00607=1096.957,64.312,441.879,176.182,16.057,152.191
C00608=1096.962,64.562,441.863,176.185,16.058,152.191
C00609=1096.968,64.811,441.847,176.187,16.059,152.191
C00610=1096.974,65.061,441.830,176.190,16.059,152.191
C00611=1096.980,65.310,441.814,176.191,16.060,152.190
C00612=1096.985,65.560,441.797,176.194,16.061,152.190
C00613=1096.991,65.809,441.781,176.196,16.062,152.190
C00614=1096.997,66.058,441.764,176.199,16.063,152.189
C00615=1097.002,66.307,441.747,176.201,16.063,152.189
C00616=1097.008,66.557,441.731,176.203,16.064,152.189
C00617=1097.013,66.806,441.714,176.206,16.065,152.188
C00618=1097.019,67.056,441.697,176.208,16.065,152.188
C00619=1097.025,67.305,441.681,176.211,16.066,152.188
C00620=1097.031,67.555,441.664,176.213,16.067,152.187
C00621=1097.036,67.804,441.647,176.216,16.068,152.187
C00622=1097.042,68.053,441.631,176.218,16.069,152.187
C00623=1097.047,68.303,441.614,176.221,16.069,152.186
C00624=1097.053,68.552,441.597,176.222,16.070,152.186
C00625=1097.059,68.801,441.580,176.225,16.071,152.185
C00626=1097.065,69.050,441.564,176.227,16.072,152.185
C00627=1097.071,69.300,441.547,176.230,16.072,152.185
C00628=1097.076,69.549,441.531,176.232,16.073,152.185
C00629=1097.082,69.798,441.514,176.234,16.073,152.184
C00630=1097.088,70.049,441.496,176.237,16.075,152.184
C00631=1097.093,70.298,441.479,176.239,16.075,152.183
C00632=1097.099,70.547,441.463,176.242,16.076,152.183
C00633=1097.105,70.797,441.446,176.244,16.076,152.183
C00634=1097.110,71.046,441.429,176.247,16.078,152.182
C00635=1097.116,71.295,441.412,176.249,16.078,152.182
C00636=1097.122,71.544,441.396,176.252,16.079,152.182
C00637=1097.127,71.794,441.379,176.254,16.080,152.181
C00638=1097.133,72.043,441.361,176.256,16.080,152.181
C00639=1097.139,72.292,441.345,176.259,16.081,152.181
C00640=1097.144,72.542,441.328,176.261,16.081,152.180
C00641=1097.150,72.791,441.311,176.264,16.083,152.180
C00642=1097.155,73.040,441.294,176.266,16.083,152.180
C00643=1097.161,73.289,441.277,176.268,16.084,152.179
C00644=1097.167,73.539,441.260,176.271,16.084,152.179
C00645=1097.173,73.789,441.243,176.274,16.085,152.179
C00646=1097.178,74.038,441.226,176.275,16.086,152.178
C00647=1097.184,74.288,441.209,176.278,16.087,152.178
C00648=1097.190,74.537,441.192,176.280,16.087,152.178
C00649=1097.195,74.786,441.175,176.283,16.088,152.177
C00650=1097.201,75.035,441.158,176.286,16.089,152.177
C00651=1097.206,75.285,441.141,176.288,16.090,152.176
C00652=1097.212,75.534,441.124,176.290,16.090,152.176
C00653=1097.218,75.784,441.107,176.293,16.090,152.176
C00654=1097.224,76.033,441.089,176.295,16.092,152.175
C00655=1097.229,76.282,441.073,176.297,16.092,152.175
C00656=1097.235,76.531,441.056,176.300,16.093,152.175
C00657=1097.241,76.781,441.039,176.302,16.093,152.174
C00658=1097.246,77.030,441.021,176.305,16.094,152.174
C00659=1097.253,77.280,441.005,176.307,16.094,152.173
C00660=1097.258,77.529,440.987,176.310,16.096,152.173
C00661=1097.263,77.779,440.970,176.312,16.096,152.173
C00662=1097.269,78.028,440.953,176.315,16.097,152.172
C00663=1097.275,78.276,440.936,176.317,16.097,152.172
C00664=1097.280,78.526,440.919,176.320,16.098,152.172
C00665=1097.286,78.776,440.901,176.322,16.099,152.171
C00666=1097.292,79.025,440.884,176.325,16.099,152.171
C00667=1097.297,79.274,440.866,176.327,16.100,152.171
C00668=1097.304,79.549,440.848,176.330,16.101,152.170
C00669=1097.310,79.823,440.829,176.333,16.102,152.170
C00670=1097.316,80.098,440.809,176.335,16.102,152.169
C00671=1097.322,80.371,440.790,176.338,16.103,152.169
C00672=1097.328,80.621,440.773,176.341,16.104,152.168
C00673=1097.333,80.870,440.756,176.343,16.104,152.168
C00674=1097.339,81.119,440.738,176.346,16.105,152.168
C00675=1097.345,81.369,440.722,176.348,16.106,152.167
C00676=1097.350,81.618,440.704,176.351,16.106,152.167
C00677=1097.356,81.867,440.686,176.353,16.107,152.167
C00678=1097.362,82.117,440.669,176.356,16.108,152.166
C00679=1097.367,82.366,440.652,176.358,16.108,152.166
C00680=1097.373,82.615,440.634,176.361,16.109,152.165
C00681=1097.378,82.864,440.617,176.363,16.110,152.165
C00682=1097.384,83.115,440.600,176.366,16.111,152.165
C00683=1097.389,83.364,440.582,176.368,16.111,152.164
C00684=1097.395,83.613,440.564,176.371,16.112,152.164
C00685=1097.401,83.862,440.547,176.374,16.112,152.163
C00686=1097.407,84.111,440.530,176.377,16.113,152.163
C00687=1097.413,84.361,440.513,176.378,16.113,152.163
C00688=1097.418,84.610,440.495,176.381,16.114,152.162
C00689=1097.424,84.859,440.478,176.384,16.114,152.162
C00690=1097.430,85.109,440.460,176.387,16.115,152.162
C00691=1097.435,85.358,440.442,176.389,16.116,152.161
C00692=1097.441,85.607,440.424,176.392,16.116,152.161
C00693=1097.447,85.857,440.407,176.394,16.117,152.160
C00694=1097.452,86.106,440.390,176.397,16.118,152.160
C00695=1097.458,86.355,440.372,176.399,16.118,152.160
C00696=1097.464,86.605,440.354,176.402,16.119,152.159
C00697=1097.469,86.854,440.337,176.404,16.119,152.159
C00698=1097.475,87.103,440.319,176.407,16.120,152.158
C00699=1097.480,87.352,440.301,176.409,16.120,152.158
C00700=1097.486,87.602,440.284,176.412,16.121,152.158
C00701=1097.492,87.851,440.266,176.414,16.121,152.157
C00702=1097.497,88.100,440.248,176.417,16.122,152.157
C00703=1097.503,88.350,440.231,176.419,16.123,152.156
C00704=1097.509,88.599,440.214,176.422,16.123,152.156
C00705=1097.514,88.848,440.196,176.425,16.124,152.155
C00706=1097.520,89.098,440.178,176.427,16.124,152.155
C00707=1097.526,89.347,440.161,176.430,16.125,152.155
C00708=1097.532,89.597,440.143,176.433,16.126,152.154
C00709=1097.538,89.846,440.125,176.435,16.126,152.154
C00710=1097.543,90.095,440.107,176.438,16.127,152.153
C00711=1097.549,90.345,440.090,176.440,16.127,152.153
C00712=1097.555,90.594,440.072,176.443,16.128,152.153
C00713=1097.561,90.842,440.054,176.445,16.128,152.152
C00714=1097.567,91.092,440.036,176.448,16.129,152.152
C00715=1097.571,91.341,440.018,176.450,16.129,152.151
C00716=1097.578,91.591,440.000,176.453,16.130,152.151
C00717=1097.583,91.840,439.982,176.455,16.130,152.150
C00718=1097.589,92.089,439.965,176.458,16.131,152.150
C00719=1097.595,92.339,439.947,176.461,16.131,152.150
C00720=1097.600,92.588,439.928,176.464,16.132,152.149
C00721=1097.605,92.837,439.911,176.466,16.132,152.149
C00722=1097.611,93.087,439.893,176.469,16.133,152.148
C00723=1097.617,93.336,439.875,176.471,16.133,152.148
C00724=1097.622,93.585,439.857,176.474,16.134,152.148
C00725=1097.628,93.834,439.839,176.476,16.134,152.147
C00726=1097.633,94.083,439.821,176.479,16.135,152.147
C00727=1097.640,94.333,439.803,176.482,16.136,152.146
C00728=1097.645,94.582,439.786,176.484,16.136,152.146
C00729=1097.650,94.831,439.767,176.487,16.137,152.145
C00730=1097.656,95.081,439.749,176.490,16.137,152.145
C00731=1097.662,95.330,439.731,176.493,16.138,152.144
C00732=1097.668,95.604,439.711,176.495,16.138,152.144
C00733=1097.674,95.879,439.691,176.498,16.139,152.144
C00734=1097.680,96.153,439.671,176.501,16.139,152.143
C00735=1097.686,96.427,439.651,176.504,16.140,152.143
C00736=1097.692,96.677,439.633,176.506,16.140,152.142
C00737=1097.698,96.926,439.616,176.509,16.141,152.142
C00738=1097.704,97.175,439.597,176.512,16.141,152.141
C00739=1097.709,97.424,439.579,176.515,16.142,152.141
C00740=1097.715,97.674,439.561,176.517,16.142,152.140
C00741=1097.721,97.923,439.543,176.520,16.143,152.140
C00742=1097.726,98.172,439.525,176.523,16.144,152.139
C00743=1097.732,98.422,439.507,176.525,16.144,152.139
C00744=1097.737,98.671,439.489,176.528,16.144,152.138
C00745=1097.743,98.920,439.470,176.530,16.145,152.138
C00746=1097.749,99.169,439.452,176.533,16.146,152.138
C00747=1097.755,99.418,439.434,176.536,16.146,152.137
C00748=1097.760,99.668,439.415,176.539,16.146,152.137
C00749=1097.766,99.917,439.398,176.541,16.146,152.136
C00750=1097.772,100.166,439.379,176.544,16.147,152.136
C00751=1097.777,100.416,439.361,176.546,16.148,152.135
C00752=1097.783,100.666,439.343,176.549,16.148,152.135
C00753=1097.789,100.914,439.325,176.552,16.148,152.134
C00754=1097.794,101.164,439.306,176.555,16.149,152.134
C00755=1097.800,101.412,439.288,176.558,16.149,152.133
C00756=1097.806,101.662,439.269,176.560,16.150,152.133
C00757=1097.811,101.911,439.251,176.563,16.151,152.133
C00758=1097.818,102.161,439.233,176.565,16.151,152.132
C00759=1097.823,102.409,439.214,176.568,16.151,152.132
C00760=1097.829,102.659,439.196,176.571,16.151,152.131
C00761=1097.834,102.908,439.177,176.574,16.152,152.131
C00762=1097.839,103.158,439.159,176.576,16.152,152.130
C00763=1097.845,103.406,439.140,176.579,16.153,152.130
C00764=1097.850,103.656,439.122,176.581,16.153,152.129
C00765=1097.856,103.905,439.104,176.584,16.154,152.129
C00766=1097.862,104.155,439.085,176.587,16.154,152.128
C00767=1097.868,104.403,439.067,176.590,16.155,152.128
C00768=1097.873,104.653,439.048,176.593,16.155,152.128
C00769=1097.879,104.902,439.030,176.595,16.155,152.127
C00770=1097.884,105.152,439.012,176.598,16.156,152.127
C00771=1097.891,105.401,438.993,176.600,16.156,152.126
C00772=1097.896,105.650,438.974,176.604,16.157,152.126
C00773=1097.902,105.899,438.956,176.607,16.158,152.125
C00774=1097.907,106.148,438.937,176.609,16.158,152.125
C00775=1097.912,106.398,438.919,176.612,16.158,152.124
C00776=1097.919,106.647,438.900,176.614,16.158,152.124
C00777=1097.924,106.896,438.881,176.617,16.159,152.123
C00778=1097.930,107.146,438.863,176.620,16.159,152.123
C00779=1097.935,107.394,438.844,176.623,16.160,152.122
C00780=1097.941,107.644,438.825,176.625,16.160,152.122
C00781=1097.947,107.894,438.807,176.628,16.161,152.121
C00782=1097.952,108.142,438.788,176.631,16.161,152.121
C00783=1097.958,108.392,438.770,176.633,16.161,152.120
C00784=1097.964,108.642,438.751,176.637,16.162,152.120
C00785=1097.969,108.890,438.732,176.639,16.162,152.119
C00786=1097.975,109.139,438.714,176.642,16.162,152.119
C00787=1097.980,109.388,438.695,176.644,16.163,152.118
C00788=1097.986,109.638,438.677,176.648,16.163,152.118
C00789=1097.992,109.887,438.657,176.651,16.164,152.117
C00790=1097.997,110.136,438.639,176.653,16.164,152.117
C00791=1098.004,110.385,438.620,176.656,16.164,152.116
C00792=1098.009,110.635,438.601,176.659,16.164,152.116
C00793=1098.015,110.885,438.582,176.661,16.165,152.115
C00794=1098.020,111.133,438.564,176.664,16.165,152.115
C00795=1098.026,111.383,438.545,176.667,16.165,152.114
C00796=1098.033,111.657,438.524,176.670,16.166,152.114
C00797=1098.038,111.931,438.503,176.673,16.167,152.113
C00798=1098.045,112.206,438.482,176.676,16.166,152.113
C00799=1098.051,112.480,438.462,176.679,16.167,152.112
C00800=1098.057,112.729,438.443,176.682,16.168,152.112
C00801=1098.062,112.979,438.424,176.685,16.167,152.111
C00802=1098.067,113.227,438.405,176.688,16.168,152.111
C00803=1098.074,113.476,438.386,176.691,16.169,152.110
C00804=1098.080,113.726,438.367,176.693,16.168,152.110
C00805=1098.085,113.975,438.348,176.696,16.169,152.109
C00806=1098.090,114.224,438.329,176.699,16.169,152.109
C00807=1098.096,114.474,438.310,176.702,16.170,152.108
C00808=1098.102,114.723,438.291,176.704,16.170,152.108
C00809=1098.107,114.972,438.273,176.708,16.170,152.107
C00810=1098.113,115.221,438.254,176.711,16.171,152.107
C00811=1098.119,115.471,438.235,176.713,16.171,152.106
C00812=1098.124,115.720,438.216,176.716,16.172,152.106
C00813=1098.129,115.969,438.196,176.718,16.171,152.105
C00814=1098.135,116.218,438.177,176.721,16.172,152.105
C00815=1098.140,116.467,438.158,176.725,16.173,152.104
C00816=1098.146,116.717,438.139,176.727,16.172,152.103
C00817=1098.152,116.966,438.120,176.730,16.173,152.103
C00818=1098.157,117.215,438.101,176.733,16.173,152.103
C00819=1098.162,117.464,438.082,176.736,16.174,152.102
C00820=1098.168,117.714,438.062,176.739,16.174,152.101
C00821=1098.174,117.962,438.042,176.741,16.174,152.101
C00822=1098.180,118.212,438.023,176.745,16.175,152.100
C00823=1098.185,118.461,438.004,176.747,16.175,152.100
C00824=1098.190,118.710,437.985,176.750,16.175,152.099
C00825=1098.196,118.959,437.966,176.753,16.176,152.099
C00826=1098.202,119.209,437.947,176.755,16.176,152.098
C00827=1098.207,119.458,437.928,176.759,16.176,152.098
C00828=1098.213,119.707,437.908,176.761,16.176,152.097
C00829=1098.218,119.957,437.889,176.764,16.177,152.097
C00830=1098.224,120.205,437.869,176.767,16.177,152.096
C00831=1098.229,120.454,437.850,176.770,16.177,152.096
C00832=1098.235,120.703,437.831,176.773,16.178,152.095
C00833=1098.241,120.953,437.812,176.775,16.178,152.095
C00834=1098.246,121.202,437.793,176.779,16.178,152.094
C00835=1098.252,121.451,437.773,176.782,16.179,152.094
C00836=1098.258,121.701,437.753,176.784,16.178,152.093
C00837=1098.263,121.949,437.735,176.788,16.179,152.092
C00838=1098.269,122.199,437.715,176.790,16.179,152.092
C00839=1098.275,122.448,437.696,176.793,16.179,152.091
C00840=1098.281,122.697,437.676,176.796,16.180,152.091
C00841=1098.286,122.946,437.657,176.799,16.180,152.090
C00842=1098.292,123.196,437.638,176.802,16.180,152.090
C00843=1098.297,123.444,437.618,176.805,16.180,152.089
C00844=1098.303,123.693,437.599,176.808,16.181,152.089
C00845=1098.309,123.943,437.580,176.811,16.181,152.088
C00846=1098.314,124.193,437.560,176.813,16.181,152.088
C00847=1098.320,124.441,437.540,176.817,16.181,152.087
C00848=1098.325,124.691,437.521,176.819,16.181,152.086
C00849=1098.331,124.940,437.501,176.822,16.182,152.086
C00850=1098.337,125.189,437.481,176.826,16.182,152.085
C00851=1098.343,125.439,437.462,176.828,16.182,152.085
C00852=1098.348,125.687,437.443,176.831,16.182,152.084
C00853=1098.354,125.936,437.423,176.835,16.183,152.084
C00854=1098.359,126.185,437.404,176.837,16.182,152.083
C00855=1098.365,126.435,437.383,176.840,16.183,152.082
C00856=1098.370,126.684,437.364,176.842,16.183,152.082
C00857=1098.376,126.933,437.344,176.846,16.183,152.081
C00858=1098.382,127.182,437.325,176.849,16.184,152.081
C00859=1098.388,127.432,437.306,176.851,16.184,152.080
C00860=1098.394,127.706,437.284,176.855,16.184,152.080
C00861=1098.400,127.980,437.262,176.858,16.184,152.079
C00862=1098.406,128.255,437.240,176.862,16.184,152.078
C00863=1098.414,128.529,437.219,176.865,16.184,152.078
C00864=1098.419,128.778,437.199,176.868,16.184,152.077
C00865=1098.425,129.027,437.179,176.871,16.185,152.077
C00866=1098.430,129.276,437.160,176.874,16.185,152.076
C00867=1098.436,129.525,437.140,176.877,16.185,152.075
C00868=1098.442,129.775,437.120,176.880,16.185,152.075
C00869=1098.447,130.024,437.100,176.882,16.185,152.074
C00870=1098.453,130.273,437.081,176.886,16.185,152.074
C00871=1098.459,130.522,437.061,176.889,16.186,152.073
C00872=1098.465,130.771,437.041,176.892,16.185,152.072
C00873=1098.471,131.020,437.022,176.895,16.186,152.072
C00874=1098.476,131.269,437.001,176.897,16.185,152.071
C00875=1098.481,131.519,436.982,176.901,16.186,152.071
C00876=1098.487,131.768,436.962,176.904,16.186,152.070
C00877=1098.493,132.017,436.942,176.906,16.186,152.070
C00878=1098.499,132.266,436.923,176.910,16.186,152.069
C00879=1098.504,132.515,436.902,176.913,16.186,152.068
C00880=1098.510,132.764,436.882,176.916,16.186,152.068
C00881=1098.515,133.014,436.862,176.919,16.187,152.067
C00882=1098.521,133.262,436.842,176.922,16.187,152.067
C00883=1098.527,133.511,436.822,176.925,16.187,152.066
C00884=1098.532,133.761,436.802,176.928,16.187,152.065
C00885=1098.538,134.010,436.783,176.930,16.187,152.065
C00886=1098.544,134.259,436.762,176.934,16.188,152.064
C00887=1098.549,134.508,436.743,176.937,16.188,152.064
C00888=1098.555,134.757,436.723,176.940,16.187,152.063
C00889=1098.560,135.006,436.702,176.943,16.188,152.062
C00890=1098.566,135.255,436.682,176.946,16.188,152.062
C00891=1098.571,135.505,436.662,176.949,16.188,152.061
C00892=1098.577,135.754,436.642,176.952,16.188,152.061
C00893=1098.583,136.003,436.622,176.956,16.188,152.060
C00894=1098.589,136.252,436.602,176.958,16.188,152.059
C00895=1098.594,136.501,436.581,176.961,16.189,152.059
C00896=1098.600,136.751,436.562,176.964,16.188,152.058
C00897=1098.606,137.000,436.542,176.967,16.189,152.058
C00898=1098.611,137.249,436.521,176.971,16.189,152.057
C00899=1098.617,137.498,436.501,176.973,16.189,152.056
C00900=1098.623,137.747,436.481,176.976,16.189,152.056
C00901=1098.629,137.996,436.461,176.980,16.189,152.055
C00902=1098.634,138.245,436.440,176.982,16.189,152.055
C00903=1098.640,138.494,436.420,176.986,16.189,152.054
C00904=1098.645,138.743,436.400,176.989,16.190,152.053
C00905=1098.651,138.992,436.380,176.992,16.189,152.053
C00906=1098.657,139.242,436.360,176.995,16.189,152.052
C00907=1098.662,139.491,436.339,176.998,16.190,152.052
C00908=1098.668,139.740,436.319,177.001,16.189,152.051
C00909=1098.673,139.989,436.298,177.004,16.190,152.050
C00910=1098.679,140.238,436.279,177.007,16.190,152.050
C00911=1098.684,140.487,436.258,177.010,16.189,152.049
C00912=1098.690,140.736,436.238,177.013,16.190,152.048
C00913=1098.696,140.986,436.217,177.016,16.190,152.048
C00914=1098.702,141.235,436.197,177.019,16.190,152.047
C00915=1098.708,141.483,436.177,177.023,16.190,152.046
C00916=1098.713,141.733,436.156,177.025,16.190,152.046
C00917=1098.718,141.982,436.135,177.029,16.190,152.045
C00918=1098.724,142.231,436.116,177.032,16.190,152.045
C00919=1098.729,142.480,436.095,177.035,16.190,152.044
C00920=1098.735,142.729,436.074,177.038,16.190,152.043
C00921=1098.741,142.978,436.054,177.041,16.190,152.043
C00922=1098.746,143.227,436.034,177.044,16.190,152.042
C00923=1098.752,143.477,436.013,177.047,16.190,152.041
C00924=1098.758,143.751,435.991,177.051,16.191,152.041
C00925=1098.764,144.025,435.968,177.054,16.191,152.040
C00926=1098.771,144.299,435.945,177.058,16.191,152.039
C00927=1098.778,144.573,435.922,177.061,16.191,152.039
C00928=1098.783,144.822,435.902,177.064,16.190,152.038
C00929=1098.788,145.071,435.881,177.067,16.190,152.037
C00930=1098.793,145.320,435.861,177.071,16.191,152.037
C00931=1098.800,145.570,435.840,177.073,16.190,152.036
C00932=1098.805,145.819,435.820,177.077,16.191,152.036
C00933=1098.811,146.067,435.798,177.080,16.191,152.035
C00934=1098.817,146.316,435.778,177.083,16.190,152.034
C00935=1098.823,146.566,435.758,177.086,16.190,152.034
C00936=1098.828,146.815,435.737,177.090,16.191,152.033
C00937=1098.833,147.064,435.716,177.092,16.190,152.032
C00938=1098.839,147.312,435.696,177.096,16.191,152.032
C00939=1098.845,147.562,435.675,177.099,16.191,152.031
C00940=1098.851,147.811,435.654,177.102,16.190,152.030
C00941=1098.856,148.060,435.633,177.105,16.190,152.030
C00942=1098.861,148.309,435.612,177.108,16.191,152.029
C00943=1098.868,148.558,435.592,177.111,16.190,152.028
C00944=1098.873,148.807,435.571,177.114,16.191,152.028
C00945=1098.879,149.056,435.550,177.118,16.191,152.027
C00946=1098.884,149.305,435.530,177.122,16.190,152.026
C00947=1098.890,149.554,435.508,177.124,16.190,152.026
C00948=1098.895,149.804,435.488,177.128,16.190,152.025
C00949=1098.901,150.053,435.467,177.131,16.191,152.024
C00950=1098.907,150.302,435.445,177.134,16.190,152.024
C00951=1098.912,150.551,435.425,177.137,16.191,152.023
C00952=1098.918,150.800,435.405,177.140,16.191,152.022
C00953=1098.924,151.049,435.383,177.143,16.190,152.022
C00954=1098.929,151.298,435.363,177.146,16.190,152.021
C00955=1098.935,151.547,435.341,177.150,16.190,152.020
C00956=1098.940,151.796,435.321,177.153,16.190,152.020
C00957=1098.946,152.045,435.299,177.156,16.190,152.019
C00958=1098.952,152.294,435.279,177.160,16.190,152.018
C00959=1098.957,152.543,435.257,177.162,16.190,152.018
C00960=1098.963,152.792,435.236,177.166,16.190,152.017
C00961=1098.968,153.042,435.216,177.169,16.190,152.016
C00962=1098.974,153.290,435.195,177.172,16.190,152.016
C00963=1098.980,153.539,435.173,177.175,16.190,152.015
C00964=1098.985,153.788,435.152,177.179,16.190,152.014
C00965=1098.992,154.038,435.131,177.182,16.190,152.014
C00966=1098.997,154.287,435.110,177.185,16.190,152.013
C00967=1099.002,154.535,435.089,177.188,16.189,152.012
C00968=1099.008,154.785,435.068,177.192,16.189,152.012
C00969=1099.014,155.034,435.047,177.194,16.189,152.011
C00970=1099.019,155.283,435.026,177.198,16.189,152.010
C00971=1099.025,155.532,435.005,177.201,16.189,152.010
C00972=1099.031,155.780,434.983,177.204,16.189,152.009
C00973=1099.037,156.030,434.962,177.207,16.189,152.008
C00974=1099.042,156.279,434.941,177.211,16.189,152.008
C00975=1099.048,156.527,434.920,177.214,16.188,152.007
C00976=1099.054,156.777,434.899,177.217,16.188,152.006
C00977=1099.058,157.026,434.877,177.221,16.189,152.006
C00978=1099.064,157.276,434.856,177.224,16.189,152.005
C00979=1099.070,157.524,434.835,177.227,16.188,152.004
C00980=1099.075,157.773,434.814,177.231,16.188,152.003
C00981=1099.082,158.022,434.792,177.234,16.189,152.003
C00982=1099.087,158.271,434.771,177.237,16.188,152.002
C00983=1099.093,158.520,434.750,177.240,16.188,152.001
C00984=1099.098,158.769,434.728,177.244,16.188,152.001
C00985=1099.104,159.019,434.707,177.246,16.187,152.000
C00986=1099.109,159.267,434.686,177.250,16.187,151.999
C00987=1099.115,159.517,434.664,177.253,16.188,151.999
C00988=1099.121,159.790,434.641,177.257,16.187,151.998
C00989=1099.127,160.064,434.617,177.261,16.187,151.997
C00990=1099.133,160.338,434.593,177.264,16.187,151.996
C00991=1099.140,160.612,434.569,177.268,16.187,151.996
C00992=1099.145,160.861,434.549,177.271,16.187,151.995
C00993=1099.151,161.110,434.527,177.274,16.187,151.994
C00994=1099.157,161.359,434.506,177.278,16.187,151.993
C00995=1099.163,161.608,434.484,177.281,16.187,151.993
C00996=1099.168,161.857,434.463,177.284,16.186,151.992
C00997=1099.174,162.106,434.441,177.287,16.186,151.991
C00998=1099.179,162.355,434.420,177.291,16.186,151.991
C00999=1099.185,162.605,434.398,177.294,16.187,151.990
C01000=1099.190,162.853,434.377,177.297,16.186,151.989
C01001=1099.195,163.102,434.355,177.301,16.186,151.989
C01002=1099.201,163.351,434.333,177.304,16.186,151.988
C01003=1099.206,163.600,434.311,177.307,16.185,151.987
C01004=1099.212,163.849,434.290,177.311,16.185,151.986
C01005=1099.218,164.098,434.269,177.314,16.186,151.986
C01006=1099.223,164.347,434.246,177.317,16.186,151.985
C01007=1099.229,164.596,434.225,177.320,16.185,151.984
C01008=1099.234,164.845,434.203,177.324,16.185,151.984
C01009=1099.240,165.094,434.182,177.327,16.185,151.983
C01010=1099.245,165.343,434.159,177.331,16.185,151.982
C01011=1099.251,165.592,434.138,177.334,16.185,151.981
C01012=1099.256,165.841,434.116,177.337,16.185,151.981
C01013=1099.262,166.090,434.095,177.341,16.185,151.980
C01014=1099.267,166.339,434.072,177.343,16.184,151.979
C01015=1099.273,166.588,434.051,177.347,16.184,151.979
C01016=1099.278,166.837,434.029,177.350,16.184,151.978
C01017=1099.284,167.086,434.008,177.354,16.185,151.977
C01018=1099.289,167.335,433.985,177.357,16.184,151.977
C01019=1099.295,167.584,433.964,177.360,16.184,151.976
C01020=1099.300,167.833,433.942,177.364,16.184,151.975
C01021=1099.307,168.082,433.919,177.367,16.184,151.974
C01022=1099.311,168.331,433.898,177.370,16.183,151.974
C01023=1099.318,168.580,433.876,177.374,16.183,151.973
C01024=1099.322,168.829,433.854,177.377,16.183,151.972
C01025=1099.329,169.078,433.832,177.381,16.183,151.971
C01026=1099.333,169.327,433.811,177.384,16.182,151.971
C01027=1099.340,169.575,433.788,177.387,16.182,151.970
C01028=1099.345,169.825,433.766,177.391,16.182,151.969
C01029=1099.351,170.073,433.745,177.394,16.182,151.968
C01030=1099.356,170.323,433.723,177.397,16.182,151.968
C01031=1099.361,170.572,433.701,177.401,16.182,151.967
C01032=1099.368,170.820,433.678,177.404,16.182,151.966
C01033=1099.373,171.070,433.656,177.407,16.181,151.966
C01034=1099.379,171.318,433.635,177.411,16.181,151.965
C01035=1099.384,171.567,433.612,177.414,16.181,151.964
C01036=1099.390,171.816,433.590,177.418,16.181,151.963
C01037=1099.395,172.065,433.568,177.421,16.180,151.963
C01038=1099.401,172.315,433.546,177.424,16.180,151.962
C01039=1099.407,172.563,433.524,177.428,16.180,151.961
C01040=1099.412,172.812,433.502,177.431,16.180,151.960
C01041=1099.418,173.061,433.480,177.434,16.180,151.960
C01042=1099.424,173.310,433.457,177.438,16.179,151.959
C01043=1099.429,173.559,433.435,177.442,16.179,151.958
C01044=1099.435,173.808,433.413,177.445,16.179,151.957
C01045=1099.441,174.057,433.391,177.448,16.179,151.957
C01046=1099.445,174.306,433.369,177.452,16.178,151.956
C01047=1099.452,174.555,433.347,177.455,16.178,151.955
C01048=1099.457,174.804,433.324,177.459,16.178,151.954
C01049=1099.464,175.053,433.302,177.462,16.178,151.954
C01050=1099.469,175.301,433.280,177.465,16.177,151.953
C01051=1099.474,175.550,433.257,177.469,16.177,151.952
C01052=1099.481,175.825,433.233,177.473,16.177,151.951
C01053=1099.487,176.098,433.209,177.476,16.177,151.950
C01054=1099.493,176.371,433.184,177.480,16.176,151.949
C01055=1099.500,176.645,433.160,177.484,16.176,151.949
C01056=1099.505,176.894,433.137,177.488,16.176,151.948
C01057=1099.510,177.142,433.115,177.491,16.176,151.947
C01058=1099.516,177.392,433.093,177.494,16.175,151.946
C01059=1099.522,177.641,433.070,177.498,16.175,151.946
C01060=1099.528,177.889,433.047,177.501,16.175,151.945
C01061=1099.534,178.139,433.026,177.505,16.175,151.944
C01062=1099.539,178.387,433.003,177.508,16.174,151.943
C01063=1099.545,178.636,432.981,177.511,16.174,151.943
C01064=1099.550,178.885,432.958,177.515,16.174,151.942
C01065=1099.557,179.134,432.935,177.519,16.174,151.941
C01066=1099.562,179.383,432.913,177.522,16.173,151.940
C01067=1099.567,179.632,432.891,177.525,16.173,151.939
C01068=1099.573,179.881,432.868,177.529,16.172,151.938
C01069=1099.579,180.130,432.846,177.533,16.172,151.938
C01070=1099.585,180.379,432.823,177.536,16.172,151.937
C01071=1099.591,180.628,432.800,177.540,16.171,151.936
C01072=1099.596,180.877,432.778,177.543,16.171,151.935
C01073=1099.603,181.126,432.756,177.547,16.171,151.935
C01074=1099.608,181.374,432.733,177.550,16.170,151.934
C01075=1099.613,181.623,432.711,177.554,16.170,151.933
C01076=1099.619,181.872,432.688,177.557,16.170,151.932
C01077=1099.625,182.121,432.665,177.561,16.169,151.931
C01078=1099.631,182.370,432.643,177.564,16.169,151.931
C01079=1099.637,182.619,432.620,177.568,16.168,151.930
C01080=1099.642,182.868,432.597,177.571,16.168,151.929
C01081=1099.648,183.117,432.574,177.575,16.168,151.928
C01082=1099.654,183.366,432.551,177.578,16.168,151.927
C01083=1099.660,183.614,432.529,177.582,16.167,151.927
C01084=1099.666,183.863,432.506,177.585,16.167,151.926
C01085=1099.671,184.113,432.484,177.589,16.167,151.925
C01086=1099.677,184.362,432.461,177.593,16.166,151.924
C01087=1099.682,184.610,432.438,177.596,16.166,151.923
C01088=1099.688,184.859,432.415,177.599,16.165,151.922
C01089=1099.694,185.107,432.393,177.603,16.165,151.922
C01090=1099.699,185.357,432.370,177.607,16.165,151.921
C01091=1099.705,185.606,432.347,177.610,16.165,151.920
C01092=1099.711,185.854,432.324,177.613,16.164,151.919
C01093=1099.717,186.103,432.301,177.617,16.164,151.919
C01094=1099.722,186.352,432.278,177.620,16.164,151.918
C01095=1099.728,186.601,432.255,177.624,16.164,151.917
C01096=1099.733,186.850,432.233,177.628,16.164,151.916
C01097=1099.739,187.099,432.210,177.631,16.163,151.915
C01098=1099.744,187.348,432.187,177.635,16.163,151.915
C01099=1099.749,187.597,432.164,177.638,16.162,151.914
C01100=1099.755,187.846,432.141,177.642,16.162,151.913
C01101=1099.761,188.095,432.118,177.646,16.162,151.912
C01102=1099.767,188.344,432.095,177.649,16.161,151.911
C01103=1099.772,188.593,432.072,177.652,16.161,151.911
C01104=1099.777,188.842,432.048,177.656,16.161,151.910
C01105=1099.783,189.090,432.025,177.660,16.160,151.909
C01106=1099.789,189.339,432.002,177.663,16.161,151.908
C01107=1099.794,189.587,431.979,177.666,16.159,151.907
C01108=1099.800,189.836,431.956,177.670,16.160,151.907
C01109=1099.805,190.085,431.933,177.674,16.159,151.906
C01110=1099.811,190.334,431.910,177.677,16.159,151.905
C01111=1099.816,190.583,431.887,177.681,16.159,151.904
C01112=1099.822,190.832,431.864,177.684,16.158,151.903
C01113=1099.827,191.081,431.840,177.688,16.158,151.903
C01114=1099.833,191.329,431.817,177.692,16.157,151.902
C01115=1099.839,191.578,431.794,177.695,16.157,151.901
C01116=1099.845,191.852,431.768,177.699,16.157,151.900
C01117=1099.851,192.125,431.743,177.703,16.157,151.899
C01118=1099.857,192.398,431.717,177.707,16.156,151.898
C01119=1099.863,192.671,431.691,177.711,16.155,151.897
C01120=1099.869,192.920,431.668,177.714,16.155,151.897
C01121=1099.875,193.169,431.645,177.718,16.155,151.896
C01122=1099.880,193.418,431.622,177.722,16.155,151.895
C01123=1099.886,193.666,431.598,177.725,16.154,151.894
C01124=1099.891,193.915,431.575,177.729,16.154,151.893
C01125=1099.897,194.164,431.552,177.733,16.153,151.892
C01126=1099.902,194.413,431.528,177.736,16.153,151.892
C01127=1099.909,194.662,431.505,177.740,16.153,151.891
C01128=1099.914,194.911,431.482,177.744,16.153,151.890
C01129=1099.921,195.160,431.458,177.747,16.152,151.889
C01130=1099.926,195.409,431.434,177.750,16.152,151.888
C01131=1099.931,195.658,431.412,177.754,16.151,151.887
C01132=1099.937,195.906,431.388,177.758,16.151,151.887
C01133=1099.942,196.155,431.364,177.762,16.151,151.886
C01134=1099.948,196.404,431.341,177.765,16.150,151.885
C01135=1099.954,196.652,431.318,177.769,16.150,151.884
C01136=1099.959,196.902,431.294,177.772,16.149,151.883
C01137=1099.966,197.151,431.270,177.776,16.149,151.883
C01138=1099.971,197.399,431.247,177.780,16.149,151.882
C01139=1099.977,197.648,431.223,177.784,16.148,151.881
C01140=1099.982,197.897,431.200,177.787,16.147,151.880
C01141=1099.988,198.146,431.176,177.791,16.147,151.879
C01142=1099.993,198.394,431.153,177.794,16.147,151.878
C01143=1099.999,198.643,431.129,177.798,16.147,151.877
C01144=1100.005,198.893,431.105,177.802,16.146,151.877
C01145=1100.011,199.141,431.082,177.805,16.145,151.876
C01146=1100.016,199.390,431.058,177.809,16.145,151.875
C01147=1100.022,199.638,431.034,177.813,16.145,151.874
C01148=1100.028,199.887,431.011,177.816,16.145,151.873
C01149=1100.034,200.137,430.987,177.820,16.144,151.872
C01150=1100.040,200.385,430.963,177.824,16.144,151.872
C01151=1100.045,200.634,430.940,177.827,16.143,151.871
C01152=1100.051,200.882,430.916,177.831,16.143,151.870
C01153=1100.056,201.132,430.892,177.834,16.142,151.869
C01154=1100.062,201.381,430.868,177.838,16.142,151.868
C01155=1100.069,201.629,430.845,177.842,16.141,151.867
C01156=1100.074,201.878,430.821,177.846,16.141,151.866
C01157=1100.080,202.126,430.797,177.849,16.140,151.865
C01158=1100.085,202.376,430.773,177.853,16.140,151.865
C01159=1100.091,202.624,430.750,177.856,16.140,151.864
C01160=1100.096,202.873,430.726,177.860,16.139,151.863
C01161=1100.103,203.121,430.702,177.864,16.139,151.862
C01162=1100.108,203.371,430.678,177.868,16.139,151.861
C01163=1100.113,203.620,430.654,177.871,16.138,151.860
C01164=1100.119,203.868,430.630,177.875,16.137,151.859
C01165=1100.125,204.117,430.606,177.879,16.137,151.859
C01166=1100.130,204.366,430.582,177.883,16.136,151.858
C01167=1100.136,204.615,430.558,177.886,16.137,151.857
C01168=1100.142,204.863,430.534,177.890,16.136,151.856
C01169=1100.147,205.112,430.510,177.894,16.136,151.855
C01170=1100.153,205.360,430.486,177.897,16.135,151.854
C01171=1100.159,205.610,430.462,177.901,16.134,151.854
C01172=1100.164,205.859,430.438,177.905,16.134,151.853
C01173=1100.170,206.107,430.414,177.908,16.134,151.852
C01174=1100.175,206.356,430.390,177.912,16.133,151.851
C01175=1100.181,206.605,430.365,177.916,16.133,151.850
C01176=1100.187,206.853,430.342,177.920,16.133,151.849
C01177=1100.192,207.102,430.318,177.923,16.132,151.848
C01178=1100.198,207.351,430.293,177.927,16.131,151.847
C01179=1100.203,207.600,430.269,177.931,16.131,151.847
C01180=1100.226,208.607,430.171,177.970,16.142,151.841
C01181=1100.235,208.976,430.135,177.975,16.143,151.840
C01182=1100.243,209.345,430.099,177.981,16.144,151.839
C01183=1100.252,209.714,430.063,177.985,16.144,151.838
C01184=1100.260,210.083,430.027,177.991,16.145,151.837
C01185=1100.266,210.332,430.002,177.994,16.145,151.837
C01186=1100.271,210.581,429.978,177.997,16.146,151.836
C01187=1100.278,210.830,429.953,178.001,16.146,151.836
C01188=1100.283,211.078,429.929,178.005,16.147,151.835
C01189=1100.288,211.327,429.904,178.008,16.148,151.834
C01190=1100.294,211.576,429.880,178.012,16.148,151.834
C01191=1100.299,211.825,429.855,178.015,16.148,151.833
C01192=1100.306,212.073,429.830,178.018,16.148,151.832
C01193=1100.311,212.322,429.806,178.022,16.149,151.832
C01194=1100.317,212.571,429.781,178.026,16.150,151.831
C01195=1100.322,212.820,429.757,178.029,16.150,151.830
C01196=1100.328,213.068,429.732,178.033,16.150,151.830
C01197=1100.334,213.317,429.707,178.036,16.151,151.829
C01198=1100.339,213.566,429.683,178.039,16.151,151.829
C01199=1100.345,213.815,429.659,178.043,16.151,151.828
C01200=1100.350,214.063,429.634,178.047,16.152,151.827
C01201=1100.356,214.312,429.609,178.050,16.153,151.827
C01202=1100.362,214.561,429.585,178.054,16.153,151.826
C01203=1100.367,214.810,429.559,178.057,16.154,151.826
C01204=1100.372,215.058,429.534,178.060,16.154,151.825
C01205=1100.378,215.307,429.510,178.064,16.155,151.824
C01206=1100.384,215.556,429.485,178.068,16.155,151.824
C01207=1100.389,215.804,429.461,178.071,16.156,151.823
C01208=1100.395,216.053,429.435,178.075,16.156,151.822
C01209=1100.401,216.301,429.411,178.078,16.156,151.822
C01210=1100.406,216.550,429.385,178.081,16.157,151.821
C01211=1100.411,216.799,429.361,178.085,16.157,151.820
C01212=1100.417,217.048,429.336,178.089,16.158,151.820
C01213=1100.423,217.296,429.311,178.092,16.158,151.819
C01214=1100.429,217.546,429.287,178.095,16.159,151.819
C01215=1100.434,217.794,429.262,178.099,16.159,151.818
C01216=1100.440,218.043,429.236,178.103,16.160,151.817
C01217=1100.446,218.292,429.211,178.106,16.160,151.817
C01218=1100.451,218.540,429.186,178.110,16.161,151.816
C01219=1100.457,218.789,429.162,178.113,16.161,151.816
C01220=1100.463,219.037,429.137,178.117,16.161,151.815
C01221=1100.468,219.287,429.111,178.121,16.162,151.814
C01222=1100.474,219.535,429.086,178.124,16.163,151.814
C01223=1100.480,219.784,429.062,178.127,16.163,151.813
C01224=1100.486,220.033,429.036,178.131,16.164,151.813
C01225=1100.491,220.281,429.011,178.135,16.164,151.812
C01226=1100.497,220.530,428.986,178.138,16.165,151.811
C01227=1100.502,220.778,428.961,178.142,16.165,151.811
C01228=1100.508,221.027,428.936,178.145,16.165,151.810
C01229=1100.514,221.276,428.911,178.148,16.166,151.809
C01230=1100.519,221.524,428.886,178.152,16.167,151.809
C01231=1100.525,221.773,428.860,178.156,16.167,151.808
C01232=1100.531,222.022,428.836,178.159,16.167,151.807
C01233=1100.539,222.395,428.797,178.165,16.168,151.807
C01234=1100.547,222.767,428.759,178.170,16.169,151.806
C01235=1100.556,223.141,428.722,178.175,16.170,151.805
C01236=1100.564,223.514,428.684,178.180,16.170,151.804
C01237=1100.570,223.762,428.658,178.184,16.172,151.803
C01238=1100.575,224.011,428.633,178.188,16.172,151.803
C01239=1100.581,224.260,428.608,178.191,16.172,151.802
C01240=1100.587,224.509,428.582,178.194,16.173,151.801
C01241=1100.592,224.757,428.557,178.198,16.174,151.801
C01242=1100.598,225.006,428.531,178.202,16.174,151.800
C01243=1100.604,225.255,428.506,178.205,16.174,151.800
C01244=1100.609,225.503,428.480,178.208,16.175,151.799
C01245=1100.615,225.752,428.455,178.212,16.176,151.798
C01246=1100.620,226.001,428.430,178.216,16.176,151.798
C01247=1100.626,226.249,428.405,178.219,16.177,151.797
C01248=1100.631,226.498,428.379,178.222,16.177,151.797
C01249=1100.637,226.747,428.354,178.227,16.178,151.796
C01250=1100.642,226.995,428.328,178.230,16.178,151.795
C01251=1100.649,227.244,428.303,178.233,16.179,151.795
C01252=1100.654,227.493,428.277,178.237,16.179,151.794
C01253=1100.660,227.741,428.251,178.241,16.180,151.794
C01254=1100.665,227.990,428.226,178.244,16.180,151.793
C01255=1100.671,228.238,428.201,178.247,16.181,151.792
C01256=1100.677,228.487,428.175,178.251,16.182,151.792
C01257=1100.683,228.736,428.149,178.255,16.182,151.791
C01258=1100.688,228.984,428.124,178.258,16.183,151.790
C01259=1100.694,229.233,428.098,178.262,16.183,151.790
C01260=1100.699,229.482,428.072,178.265,16.184,151.789
C01261=1100.706,229.730,428.046,178.269,16.185,151.789
C01262=1100.711,229.979,428.020,178.272,16.185,151.788
C01263=1100.716,230.227,427.995,178.276,16.185,151.787
C01264=1100.723,230.476,427.970,178.280,16.186,151.787
C01265=1100.728,230.725,427.944,178.283,16.187,151.786
C01266=1100.733,230.974,427.918,178.286,16.187,151.786
C01267=1100.740,231.222,427.892,178.290,16.188,151.785
C01268=1100.745,231.470,427.866,178.294,16.189,151.784
C01269=1100.750,231.719,427.840,178.297,16.189,151.784
C01270=1100.757,231.968,427.815,178.300,16.190,151.783
C01271=1100.762,232.217,427.789,178.305,16.190,151.783
C01272=1100.767,232.465,427.763,178.308,16.191,151.782
C01273=1100.773,232.713,427.737,178.311,16.192,151.782
C01274=1100.779,232.962,427.711,178.315,16.192,151.781
C01275=1100.784,233.211,427.685,178.319,16.193,151.780
C01276=1100.790,233.460,427.659,178.322,16.193,151.780
C01277=1100.796,233.708,427.633,178.326,16.194,151.779
C01278=1100.801,233.956,427.608,178.330,16.195,151.778
C01279=1100.807,234.205,427.582,178.333,16.195,151.778
C01280=1100.812,234.454,427.555,178.336,16.196,151.777
C01281=1100.818,234.703,427.529,178.340,16.197,151.777
C01282=1100.823,234.952,427.503,178.344,16.197,151.776
C01283=1100.829,235.200,427.477,178.347,16.198,151.776
C01284=1100.835,235.448,427.452,178.350,16.198,151.775
C01285=1100.843,235.813,427.413,178.355,16.199,151.774
C01286=1100.851,236.177,427.375,178.361,16.200,151.773
C01287=1100.859,236.542,427.336,178.366,16.201,151.772
C01288=1100.867,236.906,427.298,178.371,16.202,151.771
C01289=1100.873,237.155,427.273,178.375,16.203,151.771
C01290=1100.879,237.403,427.246,178.379,16.204,151.770
C01291=1100.885,237.652,427.220,178.382,16.204,151.770
C01292=1100.890,237.901,427.193,178.385,16.205,151.769
C01293=1100.896,238.150,427.167,178.389,16.206,151.769
C01294=1100.902,238.398,427.141,178.393,16.206,151.768
C01295=1100.907,238.647,427.115,178.396,16.206,151.767
C01296=1100.912,238.895,427.088,178.400,16.208,151.767
C01297=1100.918,239.143,427.062,178.403,16.208,151.766
C01298=1100.924,239.392,427.036,178.407,16.209,151.766
C01299=1100.929,239.640,427.009,178.411,16.210,151.765
C01300=1100.935,239.889,426.983,178.414,16.210,151.764
C01301=1100.941,240.138,426.957,178.417,16.211,151.764
C01302=1100.946,240.386,426.930,178.421,16.212,151.763
C01303=1100.952,240.635,426.904,178.425,16.212,151.763
C01304=1100.958,240.883,426.877,178.428,16.213,151.762
C01305=1100.963,241.132,426.851,178.432,16.214,151.762
C01306=1100.969,241.381,426.825,178.435,16.214,151.761
C01307=1100.975,241.629,426.798,178.439,16.215,151.760
C01308=1100.980,241.878,426.772,178.443,16.216,151.760
C01309=1100.986,242.126,426.745,178.446,16.216,151.759
C01310=1100.992,242.375,426.719,178.449,16.217,151.759
C01311=1100.997,242.623,426.692,178.454,16.218,151.758
C01312=1101.003,242.872,426.666,178.457,16.218,151.757
C01313=1101.009,243.120,426.639,178.460,16.219,151.757
C01314=1101.014,243.369,426.613,178.464,16.220,151.756
C01315=1101.020,243.617,426.586,178.468,16.220,151.756
C01316=1101.026,243.866,426.560,178.471,16.221,151.755
C01317=1101.031,244.114,426.533,178.475,16.222,151.755
C01318=1101.037,244.363,426.506,178.478,16.223,151.754
C01319=1101.042,244.612,426.480,178.482,16.224,151.754
C01320=1101.048,244.860,426.453,178.485,16.224,151.753
C01321=1101.054,245.109,426.426,178.489,16.224,151.752
C01322=1101.059,245.358,426.399,178.493,16.226,151.752
C01323=1101.065,245.606,426.372,178.496,16.226,151.751
C01324=1101.071,245.854,426.346,178.499,16.227,151.751
C01325=1101.077,246.103,426.319,178.503,16.228,151.750
C01326=1101.082,246.352,426.292,178.507,16.229,151.750
C01327=1101.088,246.600,426.265,178.511,16.229,151.749
C01328=1101.093,246.848,426.239,178.514,16.230,151.748
C01329=1101.099,247.097,426.212,178.517,16.231,151.748
C01330=1101.104,247.345,426.185,178.521,16.232,151.747
C01331=1101.110,247.594,426.158,178.525,16.232,151.747
C01332=1101.116,247.842,426.131,178.529,16.234,151.746
C01333=1101.121,248.091,426.104,178.532,16.234,151.746
C01334=1101.127,248.339,426.078,178.535,16.235,151.745
C01335=1101.133,248.588,426.051,178.539,16.236,151.745
C01336=1101.138,248.837,426.023,178.542,16.237,151.744
C01337=1101.146,249.194,425.985,178.548,16.237,151.743
C01338=1101.154,249.552,425.946,178.553,16.239,151.742
C01339=1101.162,249.909,425.908,178.558,16.240,151.742
C01340=1101.170,250.267,425.869,178.563,16.241,151.741
C01341=1101.175,250.516,425.841,178.566,16.242,151.740
C01342=1101.181,250.764,425.815,178.570,16.243,151.740
C01343=1101.186,251.012,425.787,178.574,16.244,151.739
C01344=1101.192,251.261,425.760,178.577,16.244,151.739
C01345=1101.198,251.510,425.732,178.581,16.245,151.738
C01346=1101.203,251.758,425.706,178.584,16.246,151.738
C01347=1101.209,252.006,425.678,178.588,16.247,151.737
C01348=1101.214,252.255,425.651,178.591,16.248,151.737
C01349=1101.219,252.503,425.624,178.595,16.249,151.736
C01350=1101.226,252.752,425.597,178.599,16.249,151.735
C01351=1101.231,253.001,425.569,178.602,16.250,151.735
C01352=1101.237,253.249,425.542,178.606,16.251,151.734
C01353=1101.242,253.498,425.515,178.609,16.252,151.734
C01354=1101.248,253.745,425.488,178.613,16.253,151.733
C01355=1101.254,253.995,425.460,178.616,16.253,151.733
C01356=1101.259,254.243,425.433,178.620,16.255,151.732
C01357=1101.265,254.491,425.405,178.624,16.255,151.732
C01358=1101.271,254.739,425.379,178.627,16.256,151.731
C01359=1101.276,254.989,425.351,178.631,16.257,151.730
C01360=1101.282,255.237,425.324,178.634,16.258,151.730
C01361=1101.287,255.485,425.297,178.638,16.259,151.729
C01362=1101.293,255.733,425.269,178.641,16.259,151.729
C01363=1101.299,255.982,425.242,178.645,16.261,151.728
C01364=1101.305,256.230,425.214,178.648,16.261,151.728
C01365=1101.310,256.479,425.187,178.652,16.262,151.727
C01366=1101.316,256.727,425.159,178.656,16.263,151.727
C01367=1101.322,256.976,425.132,178.659,16.264,151.726
C01368=1101.327,257.224,425.104,178.663,16.265,151.726
C01369=1101.333,257.472,425.077,178.666,16.266,151.725
C01370=1101.339,257.721,425.049,178.670,16.266,151.724
C01371=1101.344,257.970,425.022,178.674,16.267,151.724
C01372=1101.350,258.217,424.995,178.678,16.268,151.723
C01373=1101.356,258.467,424.967,178.681,16.269,151.723
C01374=1101.361,258.715,424.939,178.684,16.269,151.722
C01375=1101.367,258.963,424.912,178.688,16.271,151.722
C01376=1101.373,259.212,424.884,178.691,16.271,151.721
C01377=1101.379,259.460,424.857,178.695,16.272,151.721
C01378=1101.384,259.708,424.829,178.698,16.273,151.720
C01379=1101.390,259.957,424.801,178.702,16.274,151.720
C01380=1101.396,260.205,424.774,178.706,16.275,151.719
C01381=1101.401,260.453,424.746,178.710,16.276,151.719
C01382=1101.407,260.702,424.718,178.713,16.277,151.718
C01383=1101.413,260.950,424.691,178.717,16.278,151.718
C01384=1101.419,261.199,424.662,178.720,16.278,151.717
C01385=1101.424,261.447,424.635,178.724,16.280,151.716
C01386=1101.429,261.695,424.607,178.727,16.280,151.716
C01387=1101.436,261.944,424.580,178.731,16.282,151.715
C01388=1101.441,262.192,424.552,178.734,16.282,151.715
C01389=1101.449,262.547,424.512,178.740,16.284,151.714
C01390=1101.458,262.902,424.473,178.745,16.285,151.713
C01391=1101.466,263.256,424.432,178.750,16.286,151.713
C01392=1101.475,263.612,424.393,178.755,16.287,151.712
C01393=1101.480,263.860,424.365,178.758,16.288,151.711
C01394=1101.486,264.108,424.337,178.762,16.289,151.711
C01395=1101.492,264.357,424.308,178.765,16.290,151.710
C01396=1101.497,264.605,424.280,178.769,16.291,151.710
C01397=1101.503,264.854,424.252,178.773,16.292,151.709
C01398=1101.509,265.101,424.225,178.777,16.293,151.709
C01399=1101.515,265.350,424.196,178.780,16.294,151.708
C01400=1101.520,265.598,424.169,178.784,16.295,151.708
C01401=1101.526,265.847,424.141,178.787,16.295,151.707
C01402=1101.531,266.096,424.113,178.791,16.297,151.707
C01403=1101.536,266.344,424.085,178.794,16.298,151.706
C01404=1101.543,266.592,424.056,178.798,16.299,151.706
C01405=1101.548,266.840,424.028,178.801,16.300,151.705
C01406=1101.554,267.088,424.000,178.805,16.301,151.705
C01407=1101.559,267.337,423.972,178.808,16.301,151.704
C01408=1101.565,267.585,423.943,178.812,16.303,151.704
C01409=1101.571,267.833,423.915,178.815,16.304,151.703
C01410=1101.577,268.082,423.887,178.819,16.305,151.703
C01411=1101.582,268.330,423.859,178.822,16.306,151.702
C01412=1101.588,268.579,423.831,178.826,16.307,151.702
C01413=1101.593,268.827,423.803,178.830,16.307,151.701
C01414=1101.599,269.076,423.775,178.833,16.309,151.701
C01415=1101.605,269.323,423.746,178.837,16.310,151.700
C01416=1101.611,269.572,423.718,178.841,16.311,151.700
C01417=1101.616,269.820,423.690,178.845,16.312,151.699
C01418=1101.621,270.069,423.661,178.848,16.313,151.699
C01419=1101.627,270.317,423.633,178.851,16.314,151.698
C01420=1101.633,270.565,423.604,178.855,16.315,151.698
C01421=1101.639,270.814,423.575,178.859,16.316,151.697
C01422=1101.644,271.062,423.547,178.862,16.317,151.697
C01423=1101.650,271.311,423.519,178.866,16.319,151.696
C01424=1101.656,271.558,423.490,178.869,16.319,151.696
C01425=1101.662,271.807,423.462,178.873,16.320,151.695
C01426=1101.666,272.055,423.434,178.876,16.321,151.695
C01427=1101.673,272.303,423.404,178.880,16.323,151.694
C01428=1101.678,272.551,423.377,178.884,16.324,151.694
C01429=1101.684,272.800,423.348,178.887,16.325,151.693
C01430=1101.690,273.048,423.319,178.891,16.326,151.693
C01431=1101.695,273.297,423.291,178.894,16.327,151.692
C01432=1101.701,273.545,423.262,178.898,16.328,151.692
C01433=1101.706,273.793,423.234,178.901,16.329,151.691
C01434=1101.712,274.042,423.205,178.905,16.330,151.691
C01435=1101.718,274.290,423.176,178.908,16.331,151.690
C01436=1101.723,274.538,423.148,178.912,16.332,151.690
C01437=1101.729,274.786,423.119,178.916,16.334,151.690
C01438=1101.735,275.034,423.091,178.919,16.335,151.689
C01439=1101.740,275.283,423.061,178.923,16.336,151.689
C01440=1101.746,275.532,423.033,178.926,16.337,151.688
C01441=1101.754,275.888,422.992,178.931,16.338,151.687
C01442=1101.763,276.246,422.950,178.937,16.340,151.687
C01443=1101.770,276.604,422.909,178.942,16.342,151.686
C01444=1101.779,276.962,422.867,178.947,16.343,151.685
C01445=1101.784,277.210,422.838,178.950,16.344,151.685
C01446=1101.789,277.458,422.810,178.954,16.346,151.684
C01447=1101.796,277.706,422.781,178.957,16.347,151.684
C01448=1101.801,277.955,422.751,178.960,16.348,151.684
C01449=1101.807,278.203,422.723,178.964,16.349,151.683
C01450=1101.812,278.451,422.693,178.967,16.350,151.683
C01451=1101.818,278.699,422.664,178.971,16.352,151.682
C01452=1101.824,278.947,422.636,178.975,16.353,151.682
C01453=1101.829,279.196,422.607,178.978,16.354,151.681
C01454=1101.835,279.444,422.578,178.982,16.355,151.681
C01455=1101.841,279.693,422.549,178.985,16.356,151.680
C01456=1101.846,279.940,422.520,178.989,16.357,151.680
C01457=1101.852,280.189,422.490,178.993,16.359,151.680
C01458=1101.858,280.437,422.461,178.996,16.360,151.679
C01459=1101.864,280.684,422.433,179.000,16.361,151.679
C01460=1101.869,280.933,422.404,179.003,16.362,151.678
C01461=1101.875,281.182,422.375,179.007,16.364,151.678
C01462=1101.881,281.430,422.345,179.011,16.365,151.677
C01463=1101.886,281.677,422.316,179.013,16.366,151.677
C01464=1101.892,281.926,422.287,179.017,16.367,151.676
C01465=1101.897,282.175,422.258,179.021,16.369,151.676
C01466=1101.903,282.423,422.229,179.024,16.370,151.675
C01467=1101.908,282.671,422.200,179.028,16.371,151.675
C01468=1101.914,282.919,422.171,179.031,16.372,151.675
C01469=1101.920,283.167,422.141,179.035,16.374,151.674
C01470=1101.925,283.416,422.111,179.039,16.375,151.674
C01471=1101.931,283.663,422.083,179.042,16.376,151.673
C01472=1101.937,283.912,422.053,179.045,16.378,151.673
C01473=1101.942,284.160,422.023,179.049,16.379,151.672
C01474=1101.948,284.408,421.994,179.052,16.380,151.672
C01475=1101.954,284.657,421.965,179.056,16.381,151.672
C01476=1101.959,284.905,421.935,179.059,16.382,151.671
C01477=1101.965,285.153,421.906,179.063,16.384,151.671
C01478=1101.971,285.401,421.877,179.067,16.385,151.670
C01479=1101.976,285.650,421.847,179.070,16.386,151.670
C01480=1101.982,285.898,421.818,179.074,16.387,151.669
C01481=1101.987,286.145,421.789,179.077,16.389,151.669
C01482=1101.993,286.394,421.759,179.080,16.390,151.669
C01483=1101.999,286.642,421.730,179.084,16.391,151.668
C01484=1102.005,286.890,421.700,179.088,16.393,151.668
C01485=1102.010,287.138,421.670,179.091,16.394,151.667
C01486=1102.016,287.387,421.640,179.095,16.395,151.667
C01487=1102.022,287.635,421.611,179.099,16.397,151.667
C01488=1102.027,287.883,421.582,179.102,16.398,151.666
C01489=1102.032,288.131,421.553,179.106,16.399,151.666
C01490=1102.039,288.378,421.523,179.109,16.401,151.665
C01491=1102.045,288.627,421.493,179.112,16.402,151.665
C01492=1102.050,288.875,421.464,179.116,16.404,151.665
C01493=1102.058,289.242,421.419,179.121,16.405,151.664
C01494=1102.067,289.610,421.376,179.127,16.408,151.663
C01495=1102.075,289.976,421.332,179.131,16.409,151.663
C01496=1102.084,290.343,421.288,179.137,16.412,151.662
C01497=1102.089,290.591,421.258,179.140,16.413,151.662
C01498=1102.095,290.839,421.228,179.144,16.414,151.661
C01499=1102.100,291.088,421.198,179.147,16.416,151.661
C01500=1102.106,291.336,421.169,179.151,16.417,151.661
C01501=1102.112,291.584,421.138,179.154,16.418,151.660
C01502=1102.118,291.832,421.109,179.158,16.420,151.660
C01503=1102.124,292.080,421.079,179.162,16.422,151.659
C01504=1102.129,292.328,421.049,179.165,16.422,151.659
C01505=1102.135,292.577,421.020,179.169,16.424,151.659
C01506=1102.141,292.825,420.989,179.172,16.426,151.658
C01507=1102.146,293.073,420.960,179.175,16.427,151.658
C01508=1102.152,293.321,420.929,179.179,16.428,151.658
C01509=1102.157,293.569,420.900,179.183,16.430,151.657
C01510=1102.163,293.816,420.870,179.186,16.431,151.657
C01511=1102.168,294.065,420.840,179.189,16.433,151.656
C01512=1102.174,294.313,420.810,179.193,16.434,151.656
C01513=1102.180,294.560,420.779,179.197,16.436,151.656
C01514=1102.185,294.809,420.750,179.200,16.437,151.655
C01515=1102.191,295.057,420.719,179.203,16.439,151.655
C01516=1102.197,295.305,420.690,179.207,16.440,151.655
C01517=1102.203,295.553,420.659,179.211,16.442,151.654
C01518=1102.208,295.801,420.629,179.214,16.443,151.654
C01519=1102.214,296.049,420.599,179.218,16.444,151.653
C01520=1102.220,296.297,420.569,179.221,16.446,151.653
C01521=1102.225,296.546,420.540,179.224,16.447,151.653
C01522=1102.231,296.794,420.508,179.228,16.449,151.652
C01523=1102.237,297.042,420.478,179.232,16.451,151.652
C01524=1102.242,297.290,420.447,179.235,16.452,151.652
C01525=1102.248,297.538,420.418,179.238,16.453,151.651
C01526=1102.254,297.786,420.388,179.242,16.455,151.651
C01527=1102.260,298.034,420.357,179.245,16.457,151.650
C01528=1102.265,298.282,420.327,179.249,16.458,151.650
C01529=1102.270,298.531,420.297,179.252,16.460,151.650
C01530=1102.276,298.779,420.266,179.256,16.461,151.649
C01531=1102.282,299.026,420.236,179.259,16.463,151.649
C01532=1102.288,299.274,420.206,179.263,16.465,151.649
C01533=1102.293,299.522,420.175,179.267,16.466,151.648
C01534=1102.298,299.771,420.145,179.269,16.468,151.648
C01535=1102.304,300.019,420.115,179.273,16.470,151.648
C01536=1102.309,300.267,420.084,179.277,16.471,151.647
C01537=1102.315,300.515,420.053,179.280,16.473,151.647
C01538=1102.321,300.762,420.023,179.283,16.474,151.647
C01539=1102.326,301.010,419.992,179.287,16.476,151.646
C01540=1102.332,301.258,419.962,179.290,16.478,151.646
C01541=1102.338,301.506,419.931,179.294,16.480,151.646
C01542=1102.343,301.754,419.900,179.298,16.481,151.646
C01543=1102.348,302.002,419.870,179.301,16.482,151.645
C01544=1102.355,302.251,419.839,179.304,16.484,151.645
C01545=1102.363,302.631,419.793,179.309,16.487,151.644
C01546=1102.371,303.012,419.746,179.315,16.490,151.644
C01547=1102.380,303.393,419.698,179.321,16.492,151.643
C01548=1102.389,303.774,419.651,179.326,16.495,151.643
C01549=1102.395,304.022,419.621,179.329,16.496,151.643
C01550=1102.400,304.270,419.590,179.332,16.498,151.642
C01551=1102.406,304.518,419.559,179.336,16.500,151.642
C01552=1102.411,304.766,419.528,179.340,16.501,151.642
C01553=1102.416,305.014,419.498,179.343,16.503,151.642
C01554=1102.422,305.262,419.466,179.347,16.505,151.641
C01555=1102.428,305.510,419.436,179.350,16.506,151.641
C01556=1102.433,305.758,419.405,179.353,16.508,151.641
C01557=1102.439,306.006,419.374,179.357,16.510,151.640
C01558=1102.445,306.254,419.344,179.360,16.512,151.640
C01559=1102.450,306.501,419.312,179.364,16.513,151.640
C01560=1102.457,306.750,419.282,179.367,16.516,151.639
C01561=1102.462,306.998,419.251,179.370,16.517,151.639
C01562=1102.468,307.246,419.220,179.374,16.518,151.639
C01563=1102.473,307.493,419.189,179.377,16.520,151.639
C01564=1102.479,307.742,419.158,179.381,16.522,151.638
C01565=1102.485,307.990,419.127,179.385,16.524,151.638
C01566=1102.490,308.238,419.095,179.388,16.526,151.638
C01567=1102.496,308.485,419.065,179.391,16.527,151.637
C01568=1102.501,308.734,419.034,179.395,16.529,151.637
C01569=1102.508,308.981,419.003,179.398,16.531,151.637
C01570=1102.513,309.230,418.972,179.402,16.533,151.636
C01571=1102.519,309.478,418.941,179.405,16.534,151.636
C01572=1102.524,309.726,418.909,179.409,16.536,151.636
C01573=1102.530,309.973,418.879,179.412,16.537,151.636
C01574=1102.536,310.222,418.847,179.415,16.540,151.635
C01575=1102.541,310.470,418.816,179.419,16.541,151.635
C01576=1102.547,310.717,418.785,179.422,16.543,151.635
C01577=1102.553,310.966,418.754,179.426,16.545,151.634
C01578=1102.559,311.213,418.723,179.429,16.547,151.634
C01579=1102.564,311.461,418.692,179.433,16.549,151.634
C01580=1102.570,311.709,418.660,179.436,16.550,151.634
C01581=1102.576,311.957,418.629,179.439,16.552,151.633
C01582=1102.582,312.205,418.598,179.443,16.554,151.633
C01583=1102.587,312.454,418.566,179.446,16.556,151.633
C01584=1102.593,312.701,418.535,179.450,16.558,151.633
C01585=1102.599,312.950,418.504,179.453,16.559,151.632
C01586=1102.605,313.197,418.473,179.457,16.562,151.632
C01587=1102.611,313.444,418.441,179.460,16.563,151.632
C01588=1102.616,313.693,418.410,179.463,16.565,151.632
C01589=1102.622,313.940,418.379,179.467,16.567,151.631
C01590=1102.628,314.189,418.347,179.470,16.569,151.631
C01591=1102.633,314.437,418.316,179.474,16.570,151.631
C01592=1102.639,314.685,418.284,179.477,16.573,151.630
C01593=1102.645,314.932,418.253,179.481,16.574,151.630
C01594=1102.651,315.181,418.221,179.484,16.576,151.630
C01595=1102.657,315.428,418.190,179.488,16.578,151.630
C01596=1102.663,315.677,418.158,179.491,16.580,151.629
C01597=1102.670,316.059,418.109,179.496,16.584,151.629
C01598=1102.680,316.443,418.061,179.501,16.587,151.629
C01599=1102.688,316.826,418.012,179.507,16.590,151.629
C01600=1102.696,317.210,417.963,179.512,16.593,151.628
C01601=1102.702,317.458,417.931,179.515,16.595,151.628
C01602=1102.708,317.705,417.899,179.519,16.597,151.628
C01603=1102.714,317.954,417.868,179.522,16.599,151.628
C01604=1102.719,318.202,417.836,179.525,16.600,151.627
C01605=1102.725,318.450,417.804,179.528,16.603,151.627
C01606=1102.730,318.698,417.772,179.531,16.605,151.627
C01607=1102.736,318.945,417.741,179.535,16.607,151.627
C01608=1102.742,319.193,417.709,179.538,16.609,151.627
C01609=1102.747,319.441,417.677,179.542,16.611,151.626
C01610=1102.753,319.689,417.645,179.545,16.613,151.626
C01611=1102.758,319.937,417.613,179.548,16.615,151.626
C01612=1102.764,320.185,417.581,179.552,16.617,151.626
C01613=1102.769,320.433,417.549,179.555,16.619,151.626
C01614=1102.775,320.681,417.517,179.559,16.621,151.625
C01615=1102.780,320.928,417.485,179.562,16.624,151.625
C01616=1102.786,321.176,417.453,179.565,16.626,151.625
C01617=1102.792,321.424,417.422,179.569,16.628,151.625
C01618=1102.798,321.672,417.390,179.572,16.630,151.625
C01619=1102.804,321.920,417.358,179.575,16.632,151.625
C01620=1102.808,322.168,417.325,179.579,16.634,151.624
C01621=1102.814,322.416,417.293,179.582,16.636,151.624
C01622=1102.820,322.664,417.262,179.586,16.638,151.624
C01623=1102.826,322.912,417.230,179.589,16.641,151.624
C01624=1102.831,323.160,417.198,179.592,16.643,151.624
C01625=1102.837,323.407,417.165,179.596,16.645,151.624
C01626=1102.843,323.655,417.133,179.599,16.647,151.624
C01627=1102.848,323.903,417.101,179.602,16.650,151.623
C01628=1102.854,324.152,417.069,179.606,16.652,151.623
C01629=1102.859,324.399,417.037,179.609,16.654,151.623
C01630=1102.866,324.647,417.004,179.612,16.656,151.623
C01631=1102.872,324.895,416.972,179.616,16.658,151.623
C01632=1102.876,325.143,416.940,179.619,16.660,151.622
C01633=1102.882,325.391,416.908,179.622,16.662,151.622
C01634=1102.889,325.638,416.875,179.626,16.664,151.622
C01635=1102.894,325.886,416.844,179.629,16.667,151.622
C01636=1102.899,326.135,416.811,179.632,16.669,151.622
C01637=1102.906,326.382,416.778,179.636,16.671,151.622
C01638=1102.911,326.630,416.747,179.639,16.673,151.622
C01639=1102.917,326.878,416.715,179.642,16.676,151.621
C01640=1102.922,327.126,416.681,179.645,16.678,151.621
C01641=1102.928,327.373,416.650,179.649,16.680,151.621
C01642=1102.934,327.621,416.617,179.652,16.682,151.621
C01643=1102.940,327.869,416.585,179.656,16.685,151.621
C01644=1102.945,328.118,416.552,179.659,16.687,151.621
C01645=1102.951,328.364,416.520,179.662,16.689,151.621
C01646=1102.957,328.613,416.488,179.665,16.691,151.620
C01647=1102.963,328.861,416.455,179.669,16.693,151.620
C01648=1102.969,329.109,416.423,179.672,16.696,151.620
C01649=1102.977,329.485,416.373,179.677,16.699,151.620
C01650=1102.986,329.861,416.324,179.682,16.702,151.620
C01651=1102.995,330.237,416.274,179.687,16.706,151.620
C01652=1103.004,330.614,416.225,179.692,16.709,151.619
C01653=1103.010,330.861,416.192,179.696,16.712,151.619
C01654=1103.015,331.109,416.160,179.699,16.715,151.619
C01655=1103.021,331.357,416.127,179.702,16.717,151.619
C01656=1103.027,331.605,416.095,179.705,16.719,151.619
C01657=1103.033,331.853,416.061,179.709,16.721,151.619
C01658=1103.039,332.101,416.029,179.712,16.724,151.619
C01659=1103.044,332.349,415.996,179.715,16.726,151.619
C01660=1103.050,332.596,415.964,179.718,16.729,151.619
C01661=1103.055,332.844,415.930,179.722,16.731,151.619
C01662=1103.062,333.092,415.898,179.725,16.733,151.618
C01663=1103.067,333.340,415.865,179.728,16.736,151.618
C01664=1103.072,333.587,415.832,179.731,16.738,151.618
C01665=1103.078,333.835,415.799,179.735,16.741,151.618
C01666=1103.084,334.083,415.766,179.738,16.744,151.618
C01667=1103.089,334.331,415.733,179.742,16.746,151.618
C01668=1103.095,334.579,415.701,179.745,16.748,151.618
C01669=1103.100,334.826,415.668,179.748,16.751,151.618
C01670=1103.107,335.074,415.635,179.751,16.753,151.618
C01671=1103.112,335.322,415.602,179.754,16.756,151.618
C01672=1103.117,335.570,415.569,179.757,16.758,151.618
C01673=1103.124,335.818,415.536,179.761,16.761,151.618
C01674=1103.129,336.066,415.503,179.764,16.764,151.618
C01675=1103.135,336.314,415.469,179.768,16.766,151.618
C01676=1103.140,336.560,415.437,179.771,16.769,151.618
C01677=1103.146,336.808,415.404,179.774,16.771,151.618
C01678=1103.152,337.056,415.370,179.777,16.773,151.618
C01679=1103.158,337.304,415.338,179.780,16.776,151.617
C01680=1103.163,337.552,415.304,179.784,16.779,151.617
C01681=1103.169,337.800,415.271,179.787,16.782,151.617
C01682=1103.174,338.048,415.238,179.790,16.784,151.617
C01683=1103.181,338.295,415.205,179.793,16.787,151.617
C01684=1103.186,338.543,415.172,179.796,16.789,151.617
C01685=1103.192,338.791,415.138,179.800,16.791,151.617
C01686=1103.197,339.038,415.105,179.804,16.795,151.617
C01687=1103.203,339.286,415.073,179.807,16.797,151.617
C01688=1103.209,339.534,415.039,179.810,16.800,151.617
C01689=1103.214,339.782,415.006,179.813,16.802,151.617
C01690=1103.220,340.029,414.972,179.816,16.805,151.617
C01691=1103.226,340.277,414.938,179.819,16.808,151.617
C01692=1103.231,340.525,414.905,179.822,16.811,151.617
C01693=1103.237,340.773,414.872,179.826,16.813,151.617
C01694=1103.242,341.021,414.838,179.829,16.816,151.617
C01695=1103.249,341.268,414.806,179.832,16.819,151.617
C01696=1103.254,341.515,414.772,179.836,16.822,151.617
C01697=1103.260,341.763,414.738,179.839,16.824,151.617
C01698=1103.266,342.011,414.705,179.842,16.827,151.617
C01699=1103.271,342.259,414.672,179.845,16.830,151.617
C01700=1103.277,342.506,414.638,179.848,16.833,151.617
C01701=1103.286,342.877,414.588,179.853,16.837,151.617
C01702=1103.294,343.247,414.537,179.858,16.841,151.617
C01703=1103.303,343.617,414.488,179.862,16.845,151.618
C01704=1103.311,343.988,414.437,179.867,16.849,151.618
C01705=1103.316,344.235,414.403,179.870,16.852,151.618
C01706=1103.322,344.483,414.370,179.873,16.855,151.618
C01707=1103.328,344.730,414.336,179.877,16.858,151.618
C01708=1103.333,344.978,414.303,179.880,16.861,151.618
C01709=1103.339,345.226,414.269,179.883,16.863,151.618
C01710=1103.345,345.473,414.235,179.886,16.866,151.618
C01711=1103.350,345.721,414.202,179.890,16.869,151.618
C01712=1103.356,345.969,414.168,179.893,16.872,151.618
C01713=1103.362,346.216,414.134,179.896,16.875,151.618
C01714=1103.368,346.464,414.100,179.899,16.878,151.618
C01715=1103.373,346.712,414.067,179.902,16.881,151.618
C01716=1103.379,346.959,414.033,179.905,16.884,151.618
C01717=1103.385,347.206,413.999,179.908,16.886,151.618
C01718=1103.390,347.454,413.965,179.912,16.890,151.618
C01719=1103.396,347.702,413.931,179.915,16.893,151.618
C01720=1103.402,347.950,413.897,179.918,16.896,151.619
C01721=1103.408,348.198,413.863,179.921,16.899,151.619
C01722=1103.414,348.445,413.829,179.924,16.902,151.619
C01723=1103.419,348.693,413.796,179.927,16.905,151.619
C01724=1103.424,348.940,413.761,179.930,16.907,151.619
C01725=1103.430,349.188,413.727,179.934,16.911,151.619
C01726=1103.436,349.436,413.694,179.937,16.914,151.619
C01727=1103.441,349.683,413.660,179.940,16.916,151.619
C01728=1103.447,349.930,413.625,179.943,16.920,151.619
C01729=1103.453,350.179,413.591,179.946,16.923,151.620
C01730=1103.459,350.426,413.557,179.949,16.926,151.620
C01731=1103.464,350.674,413.523,179.953,16.929,151.620
C01732=1103.470,350.921,413.489,179.955,16.932,151.620
C01733=1103.475,351.169,413.455,179.958,16.935,151.620
C01734=1103.481,351.416,413.421,179.962,16.938,151.620
C01735=1103.487,351.664,413.387,179.965,16.941,151.620
C01736=1103.493,351.912,413.352,179.968,16.945,151.620
C01737=1103.498,352.159,413.318,179.971,16.948,151.620
C01738=1103.504,352.407,413.284,179.974,16.950,151.621
C01739=1103.509,352.654,413.249,179.978,16.954,151.621
C01740=1103.515,352.901,413.215,179.980,16.957,151.621
C01741=1103.522,353.149,413.181,179.983,16.960,151.621
C01742=1103.527,353.397,413.146,179.987,16.964,151.621
C01743=1103.532,353.645,413.113,179.990,16.967,151.621
C01744=1103.538,353.892,413.079,179.992,16.969,151.622
C01745=1103.543,354.140,413.044,179.996,16.973,151.622
C01746=1103.550,354.388,413.010,179.999,16.976,151.622
C01747=1103.555,354.635,412.975,-179.998,16.980,151.622
C01748=1103.561,354.883,412.941,-179.995,16.983,151.622
C01749=1103.566,355.130,412.906,-179.992,16.986,151.622
C01750=1103.572,355.377,412.872,-179.989,16.990,151.623
C01751=1103.578,355.625,412.837,-179.986,16.992,151.623
C01752=1103.584,355.873,412.803,-179.983,16.996,151.623
C01753=1103.592,356.245,412.751,-179.978,17.001,151.623
C01754=1103.601,356.617,412.699,-179.974,17.006,151.624
C01755=1103.609,356.990,412.647,-179.969,17.011,151.624
C01756=1103.618,357.363,412.595,-179.965,17.016,151.624
C01757=1103.623,357.610,412.561,-179.961,17.019,151.624
C01758=1103.630,357.858,412.525,-179.958,17.022,151.625
C01759=1103.635,358.105,412.491,-179.955,17.026,151.625
C01760=1103.640,358.352,412.457,-179.952,17.029,151.625
C01761=1103.646,358.601,412.421,-179.949,17.033,151.625
C01762=1103.652,358.847,412.387,-179.946,17.036,151.625
C01763=1103.658,359.095,412.352,-179.943,17.039,151.626
C01764=1103.663,359.342,412.318,-179.940,17.043,151.626
C01765=1103.669,359.590,412.282,-179.937,17.046,151.626
C01766=1103.675,359.838,412.248,-179.934,17.050,151.626
C01767=1103.681,360.086,412.213,-179.931,17.053,151.627
C01768=1103.686,360.332,412.178,-179.928,17.057,151.627
C01769=1103.692,360.580,412.144,-179.925,17.060,151.627
C01770=1103.698,360.827,412.108,-179.922,17.064,151.627
C01771=1103.703,361.075,412.073,-179.919,17.067,151.628
C01772=1103.709,361.323,412.039,-179.916,17.071,151.628
C01773=1103.715,361.569,412.004,-179.913,17.074,151.628
C01774=1103.720,361.818,411.969,-179.910,17.078,151.628
C01775=1103.726,362.065,411.934,-179.907,17.081,151.629
C01776=1103.732,362.313,411.899,-179.904,17.085,151.629
C01777=1103.738,362.560,411.864,-179.901,17.089,151.629
C01778=1103.743,362.807,411.829,-179.898,17.093,151.630
C01779=1103.749,363.055,411.793,-179.895,17.096,151.630
C01780=1103.755,363.302,411.759,-179.892,17.100,151.630
C01781=1103.760,363.549,411.724,-179.890,17.103,151.630
C01782=1103.766,363.797,411.688,-179.886,17.107,151.631
C01783=1103.771,364.044,411.654,-179.884,17.110,151.631
C01784=1103.777,364.292,411.618,-179.881,17.114,151.631
C01785=1103.783,364.539,411.584,-179.877,17.118,151.632
C01786=1103.789,364.786,411.549,-179.875,17.122,151.632
C01787=1103.795,365.034,411.513,-179.871,17.126,151.632
C01788=1103.800,365.282,411.478,-179.869,17.129,151.633
C01789=1103.806,365.529,411.442,-179.866,17.133,151.633
C01790=1103.811,365.776,411.407,-179.863,17.136,151.633
C01791=1103.818,366.024,411.372,-179.860,17.140,151.634
C01792=1103.823,366.271,411.337,-179.857,17.144,151.634
C01793=1103.829,366.518,411.302,-179.854,17.148,151.634
C01794=1103.835,366.766,411.266,-179.851,17.152,151.635
C01795=1103.840,367.013,411.231,-179.849,17.155,151.635
C01796=1103.846,367.260,411.195,-179.845,17.159,151.635
C01797=1103.851,367.508,411.160,-179.843,17.163,151.636
C01798=1103.857,367.756,411.125,-179.840,17.167,151.636
C01799=1103.863,368.003,411.089,-179.836,17.171,151.636
C01800=1103.869,368.250,411.054,-179.834,17.174,151.637
C01801=1103.874,368.497,411.018,-179.831,17.179,151.637
C01802=1103.880,368.744,410.983,-179.828,17.182,151.638
C01803=1103.886,368.992,410.947,-179.825,17.186,151.638
C01804=1103.891,369.239,410.912,-179.822,17.190,151.638
C01805=1103.900,369.627,410.856,-179.818,17.197,151.639
C01806=1103.909,370.014,410.800,-179.814,17.203,151.640
C01807=1103.918,370.402,410.745,-179.809,17.209,151.640
C01808=1103.926,370.789,410.689,-179.804,17.215,151.641
C01809=1103.932,371.036,410.653,-179.802,17.219,151.641
C01810=1103.938,371.283,410.618,-179.799,17.223,151.642
C01811=1103.944,371.531,410.582,-179.795,17.227,151.642
C01812=1103.949,371.778,410.546,-179.793,17.231,151.642
C01813=1103.955,372.026,410.511,-179.790,17.235,151.643
C01814=1103.961,372.273,410.475,-179.787,17.240,151.643
C01815=1103.967,372.520,410.439,-179.785,17.243,151.644
C01816=1103.972,372.768,410.403,-179.782,17.247,151.644
